KUKA KRL program: MyProgram_256().src

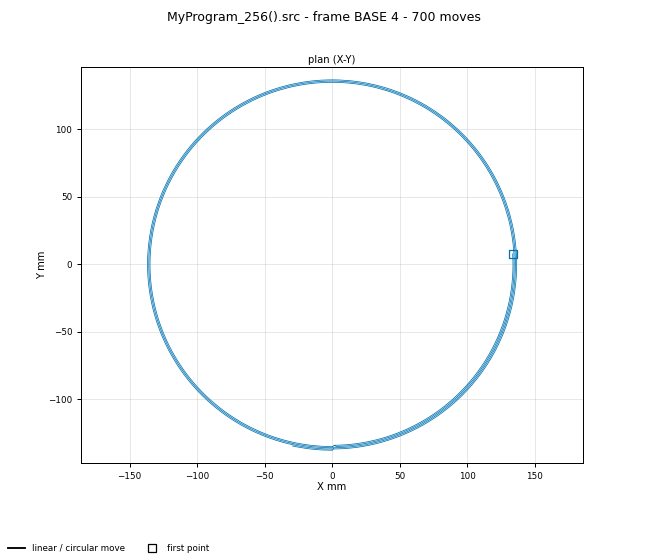
[picture p0: tool path of MyProgram_256().src in frame BASE 4, 700 of 700 moves have a stored position in this frame; points joined in program order, loops and branches not executed]
&ACCESS RVP
&REL 1
&PARAM TEMPLATE = C:\KRC\Roboter\Template\vorgabe
&PARAM EDITMASK = *
DEF MyProgram_256()
; ---- Setting reference (Base) ----
$BASE = BASE_DATA[4]

; --------------------------
; ---- Setting tool (TCP) ----
$TOOL = TOOL_DATA[3]
; --------------------------

$VEL.CP = VEL_APROX_PRINT
Startdeposition()
$VEL.CP = VEL_PRINT
LIN {X 133.7906,Y 7.8081,Z 166,A 3.583,B 11.1418,C 0.1363,E1 11.3023,E2 447.1439} C_DIS
LIN {X 133.9693,Y 3.6015,Z 166,A 1.8917,B 11.1418,C 0.1387,E1 11.3024,E2 448.8238} C_DIS
LIN {X 134.0189,Y -0.4124,Z 166,A 0.0697,B 11.1418,C 0.1466,E1 11.3024,E2 450.6604} C_DIS
LIN {X 133.9478,Y -4.3751,Z 166,A -1.598,B 11.1416,C 0.1508,E1 11.3024,E2 452.3268} C_DIS
LIN {X 133.7538,Y -8.4056,Z 166,A -3.1449,B 11.1416,C 0.1512,E1 11.3021,E2 453.8538} C_DIS
LIN {X 133.4765,Y -12.0532,Z 166,A -4.846,B 11.1416,C 0.1594,E1 11.3017,E2 455.5733} C_DIS
LIN {X 133.0684,Y -15.9212,Z 166,A -6.3681,B 11.1416,C 0.1606,E1 11.3012,E2 457.08} C_DIS
LIN {X 132.6216,Y -19.2954,Z 166,A -7.7805,B 11.1415,C 0.1637,E1 11.3007,E2 458.4888} C_DIS
LIN {X 131.994,Y -23.2035,Z 166,A -9.5019,B 11.1414,C 0.1694,E1 11.2999,E2 460.2156} C_DIS
LIN {X 131.3378,Y -26.6655,Z 166,A -10.9987,B 11.1414,C 0.1735,E1 11.2991,E2 461.7128} C_DIS
LIN {X 130.4251,Y -30.8268,Z 166,A -13.677,B 11.1409,C 0.2014,E1 11.2973,E2 464.497} C_DIS
LIN {X 128.7428,Y -37.2306,Z 166,A -15.3883,B 11.1412,C 0.18,E1 11.2961,E2 466.0757} C_DIS
LIN {X 127.5273,Y -41.2019,Z 166,A -17.6042,B 11.1409,C 0.1967,E1 11.2942,E2 468.3474} C_DIS
LIN {X 126.4482,Y -44.4042,Z 166,A -18.6879,B 11.141,C 0.1912,E1 11.2933,E2 469.3887} C_DIS
LIN {X 125.1769,Y -47.8735,Z 166,A -20.2354,B 11.141,C 0.1948,E1 11.2918,E2 470.9341} C_DIS
LIN {X 124.0766,Y -50.6551,Z 166,A -21.541,B 11.141,C 0.199,E1 11.2904,E2 472.2445} C_DIS
LIN {X 122.8258,Y -53.6156,Z 166,A -22.8653,B 11.1409,C 0.2015,E1 11.2889,E2 473.5642} C_DIS
LIN {X 120.5287,Y -58.6003,Z 166,A -25.1853,B 11.1408,C 0.2071,E1 11.2862,E2 475.8837} C_DIS
LIN {X 119.1646,Y -61.3246,Z 166,A -26.4556,B 11.1408,C 0.2098,E1 11.2846,E2 477.1515} C_DIS
LIN {X 117.7601,Y -63.9821,Z 166,A -27.884,B 11.1406,C 0.2169,E1 11.2827,E2 478.599} C_DIS
LIN {X 115.3948,Y -68.156,Z 166,A -29.8951,B 11.1405,C 0.2212,E1 11.2799,E2 480.6076} C_DIS
LIN {X 113.0597,Y -71.9634,Z 166,A -31.8065,B 11.1404,C 0.2262,E1 11.277,E2 482.5214} C_DIS
LIN {X 110.6658,Y -75.5929,Z 166,A -33.6473,B 11.1404,C 0.2303,E1 11.2742,E2 484.362} C_DIS
LIN {X 107.9816,Y -79.3793,Z 166,A -35.5798,B 11.1402,C 0.2339,E1 11.271,E2 486.2904} C_DIS
LIN {X 105.2313,Y -82.9912,Z 166,A -37.5088,B 11.1402,C 0.2382,E1 11.2677,E2 488.2202} C_DIS
LIN {X 101.0585,Y -88.0239,Z 166,A -40.4879,B 11.1399,C 0.2495,E1 11.2623,E2 491.2248} C_DIS
LIN {X 98.7885,Y -90.5647,Z 166,A -41.3605,B 11.1402,C 0.2376,E1 11.2608,E2 492.0274} C_DIS
LIN {X 93.0666,Y -96.4352,Z 166,A -44.9331,B 11.14,C 0.247,E1 11.2538,E2 495.6122} C_DIS
LIN {X 88.7789,Y -100.3962,Z 166,A -47.5027,B 11.1398,C 0.2542,E1 11.2485,E2 498.1936} C_DIS
LIN {X 83.3335,Y -104.9603,Z 166,A -50.5306,B 11.1397,C 0.2599,E1 11.242,E2 501.2236} C_DIS
LIN {X 79.6928,Y -107.7513,Z 166,A -52.6048,B 11.1395,C 0.2665,E1 11.2373,E2 503.3137} C_DIS
LIN {X 76.2597,Y -110.2074,Z 166,A -54.7708,B 11.1392,C 0.2789,E1 11.2323,E2 505.5257} C_DIS
LIN {X 72.8142,Y -112.5127,Z 166,A -56.0319,B 11.1394,C 0.269,E1 11.2295,E2 506.7259} C_DIS
LIN {X 70.1028,Y -114.2222,Z 166,A -57.527,B 11.1394,C 0.2744,E1 11.2259,E2 508.2376} C_DIS
LIN {X 66.5644,Y -116.3199,Z 166,A -59.1858,B 11.1394,C 0.2747,E1 11.2219,E2 509.8859} C_DIS
LIN {X 63.435,Y -118.0555,Z 166,A -60.712,B 11.1393,C 0.2769,E1 11.2181,E2 511.413} C_DIS
LIN {X 60.4507,Y -119.6095,Z 166,A -62.0754,B 11.1393,C 0.2771,E1 11.2148,E2 512.7684} C_DIS
LIN {X 57.3326,Y -121.1354,Z 166,A -63.5711,B 11.1392,C 0.2795,E1 11.211,E2 514.2669} C_DIS
LIN {X 54.3356,Y -122.5088,Z 166,A -64.9633,B 11.1392,C 0.2809,E1 11.2075,E2 515.6581} C_DIS
LIN {X 51.2255,Y -123.8416,Z 166,A -66.4225,B 11.1392,C 0.2831,E1 11.2037,E2 517.1201} C_DIS
LIN {X 48.4559,Y -124.9505,Z 166,A -67.7161,B 11.1391,C 0.285,E1 11.2003,E2 518.4169} C_DIS
LIN {X 44.8142,Y -126.3042,Z 166,A -69.8247,B 11.1387,C 0.298,E1 11.1947,E2 520.5818} C_DIS
LIN {X 40.9151,Y -127.6189,Z 166,A -71.2137,B 11.1389,C 0.2907,E1 11.1911,E2 521.9268} C_DIS
LIN {X 37.414,Y -128.6891,Z 166,A -73.2769,B 11.1386,C 0.3044,E1 11.1854,E2 524.052} C_DIS
LIN {X 32.597,Y -129.9931,Z 166,A -74.6609,B 11.139,C 0.2879,E1 11.1819,E2 525.3459} C_DIS
LIN {X 29.7032,Y -130.6843,Z 166,A -76.0129,B 11.139,C 0.2909,E1 11.1782,E2 526.7087} C_DIS
LIN {X 26.3148,Y -131.4091,Z 166,A -77.4611,B 11.1389,C 0.2911,E1 11.1742,E2 528.1538} C_DIS
LIN {X 23.6903,Y -131.9069,Z 166,A -78.6623,B 11.1389,C 0.2933,E1 11.1709,E2 529.363} C_DIS
LIN {X 20.3393,Y -132.4651,Z 166,A -80.0685,B 11.1389,C 0.2931,E1 11.167,E2 530.7645} C_DIS
LIN {X 16.9036,Y -132.9481,Z 166,A -81.7085,B 11.1387,C 0.2976,E1 11.1624,E2 532.4246} C_DIS
LIN {X 12.8845,Y -133.3967,Z 166,A -83.3725,B 11.1387,C 0.2968,E1 11.1578,E2 534.0817} C_DIS
LIN {X 9.0475,Y -133.7137,Z 166,A -85.082,B 11.1387,C 0.2989,E1 11.153,E2 535.8} C_DIS
LIN {X 4.8862,Y -133.9289,Z 166,A -86.7229,B 11.1387,C 0.296,E1 11.1485,E2 537.4245} C_DIS
LIN {X 0.9791,Y -134.0137,Z 166,A -87.7099,B 11.1392,C 0.28,E1 11.146,E2 538.3279} C_DIS
Enddeposition()
LIN {X 0.9791,Y -134.0137,Z 166,A -87.7099,B 11.1392,C 0.28,E1 11.146,E2 538.3279} C_DIS
Startdeposition()
$VEL.CP = VEL_PRINT
LIN {X 3.2943,Y -134.8946,Z 166,A -86.6554,B 11.0822,C 0.2874,E1 11.092,E2 537.3154} C_DIS
LIN {X 7.444,Y -134.7302,Z 166,A -84.8631,B 11.0822,C 0.2862,E1 11.097,E2 535.5186} C_DIS
LIN {X 11.3456,Y -134.4561,Z 166,A -83.3067,B 11.0822,C 0.2881,E1 11.1013,E2 533.9743} C_DIS
LIN {X 14.7948,Y -134.1208,Z 166,A -81.735,B 11.0822,C 0.285,E1 11.1057,E2 532.3891} C_DIS
LIN {X 18.5599,Y -133.6524,Z 166,A -80.1797,B 11.0822,C 0.2856,E1 11.11,E2 530.84} C_DIS
LIN {X 22.1578,Y -133.1021,Z 166,A -78.6595,B 11.0822,C 0.2853,E1 11.1142,E2 529.3219} C_DIS
LIN {X 26.1565,Y -132.3762,Z 166,A -76.8587,B 11.0823,C 0.2822,E1 11.1192,E2 527.5106} C_DIS
LIN {X 29.8744,Y -131.5852,Z 166,A -75.3332,B 11.0823,C 0.2832,E1 11.1233,E2 525.995} C_DIS
LIN {X 33.1445,Y -130.7996,Z 166,A -73.7747,B 11.0823,C 0.2787,E1 11.1276,E2 524.4191} C_DIS
LIN {X 38.4727,Y -129.334,Z 166,A -70.7758,B 11.0828,C 0.2601,E1 11.1359,E2 521.336} C_DIS
LIN {X 44.2696,Y -127.4648,Z 166,A -68.935,B 11.0825,C 0.2762,E1 11.1405,E2 519.5874} C_DIS
LIN {X 49.6533,Y -125.4682,Z 166,A -66.5654,B 11.0825,C 0.2751,E1 11.1466,E2 517.2246} C_DIS
LIN {X 53.2645,Y -123.976,Z 166,A -64.8895,B 11.0825,C 0.2726,E1 11.151,E2 515.5452} C_DIS
LIN {X 57.4577,Y -122.0912,Z 166,A -62.8633,B 11.0827,C 0.2681,E1 11.1561,E2 513.5079} C_DIS
LIN {X 61.1579,Y -120.2778,Z 166,A -61.2251,B 11.0827,C 0.2684,E1 11.1602,E2 511.8822} C_DIS
LIN {X 64.7709,Y -118.3737,Z 166,A -59.4725,B 11.0827,C 0.2653,E1 11.1645,E2 510.1257} C_DIS
LIN {X 68.6942,Y -116.1415,Z 166,A -57.6684,B 11.0827,C 0.2653,E1 11.1688,E2 508.334} C_DIS
LIN {X 72.9984,Y -113.4851,Z 166,A -55.0485,B 11.0831,C 0.2494,E1 11.1752,E2 505.6525} C_DIS
LIN {X 76.5356,Y -111.1302,Z 166,A -53.6572,B 11.0829,C 0.2569,E1 11.1783,E2 504.3116} C_DIS
LIN {X 78.8554,Y -109.4969,Z 166,A -52.2038,B 11.0831,C 0.2483,E1 11.1816,E2 502.8257} C_DIS
LIN {X 81.6626,Y -107.4193,Z 166,A -50.9427,B 11.0831,C 0.2513,E1 11.1844,E2 501.5911} C_DIS
LIN {X 85.2525,Y -104.5926,Z 166,A -49.0521,B 11.0831,C 0.2488,E1 11.1885,E2 499.7047} C_DIS
LIN {X 88.9879,Y -101.434,Z 166,A -46.5816,B 11.0834,C 0.2343,E1 11.1938,E2 497.1824} C_DIS
LIN {X 92.2495,Y -98.4766,Z 166,A -45.1583,B 11.0832,C 0.2422,E1 11.1966,E2 495.8134} C_DIS
LIN {X 97.1282,Y -93.6683,Z 166,A -42.264,B 11.0834,C 0.2363,E1 11.2023,E2 492.9179} C_DIS
LIN {X 104.1946,Y -85.7394,Z 166,A -37.7832,B 11.0836,C 0.2268,E1 11.2106,E2 488.4361} C_DIS
LIN {X 106.9401,Y -82.2894,Z 166,A -35.9194,B 11.0836,C 0.2225,E1 11.2138,E2 486.5713} C_DIS
LIN {X 109.6131,Y -78.6932,Z 166,A -34.07,B 11.0837,C 0.2193,E1 11.2168,E2 484.7265} C_DIS
LIN {X 112.0482,Y -75.1856,Z 166,A -32.2399,B 11.0838,C 0.2143,E1 11.2197,E2 482.8922} C_DIS
LIN {X 114.4423,Y -71.4883,Z 166,A -30.4055,B 11.0838,C 0.2105,E1 11.2224,E2 481.0602} C_DIS
LIN {X 116.8454,Y -67.4889,Z 166,A -28.4762,B 11.084,C 0.2068,E1 11.2251,E2 479.1352} C_DIS
LIN {X 119.0573,Y -63.5067,Z 166,A -26.6472,B 11.084,C 0.2045,E1 11.2276,E2 477.3172} C_DIS
LIN {X 120.8288,Y -60.0633,Z 166,A -25.0143,B 11.084,C 0.2004,E1 11.2296,E2 475.6837} C_DIS
LIN {X 122.3657,Y -56.8659,Z 166,A -23.4203,B 11.0842,C 0.1939,E1 11.2315,E2 474.077} C_DIS
LIN {X 124.3117,Y -52.4778,Z 166,A -21.4551,B 11.0842,C 0.1903,E1 11.2337,E2 472.1187} C_DIS
LIN {X 125.397,Y -49.8305,Z 166,A -19.8941,B 11.0845,C 0.1776,E1 11.2354,E2 470.5129} C_DIS
LIN {X 126.8018,Y -46.1359,Z 166,A -18.7424,B 11.0843,C 0.1871,E1 11.2364,E2 469.4254} C_DIS
LIN {X 128.0668,Y -42.497,Z 166,A -17.0395,B 11.0844,C 0.1807,E1 11.238,E2 467.7122} C_DIS
LIN {X 129.3159,Y -38.5344,Z 166,A -15.1809,B 11.0845,C 0.1732,E1 11.2395,E2 465.8399} C_DIS
LIN {X 131.0199,Y -32.2697,Z 166,A -12.4407,B 11.0846,C 0.1657,E1 11.2414,E2 463.0987} C_DIS
LIN {X 132.0233,Y -27.8806,Z 166,A -10.616,B 11.0846,C 0.1625,E1 11.2425,E2 461.2827} C_DIS
LIN {X 132.6854,Y -24.5424,Z 166,A -9.1493,B 11.0847,C 0.1578,E1 11.2433,E2 459.8117} C_DIS
LIN {X 133.3765,Y -20.4421,Z 166,A -7.5048,B 11.0847,C 0.1559,E1 11.244,E2 458.1803} C_DIS
LIN {X 133.9607,Y -16.1777,Z 166,A -5.7189,B 11.0848,C 0.1516,E1 11.2446,E2 456.3976} C_DIS
LIN {X 134.3488,Y -12.557,Z 166,A -4.1158,B 11.0849,C 0.1456,E1 11.2451,E2 454.7859} C_DIS
LIN {X 134.6817,Y -8.2474,Z 166,A -2.3861,B 11.0849,C 0.143,E1 11.2454,E2 453.0673} C_DIS
LIN {X 134.8728,Y -4.0791,Z 166,A -0.6094,B 11.085,C 0.1377,E1 11.2456,E2 451.2882} C_DIS
LIN {X 134.9378,Y -0.04,Z 166,A 1.162,B 11.085,C 0.1311,E1 11.2456,E2 449.5082} C_DIS
LIN {X 134.8901,Y 3.4547,Z 166,A 2.489,B 11.085,C 0.131,E1 11.2456,E2 448.199} C_DIS
LIN {X 134.7486,Y 7.0766,Z 166,A 4.1116,B 11.0852,C 0.1242,E1 11.2454,E2 446.5645} C_DIS
LIN {X 134.4614,Y 11.2831,Z 166,A 5.8418,B 11.0852,C 0.1206,E1 11.245,E2 444.8399} C_DIS
LIN {X 134.0572,Y 15.3692,Z 166,A 7.6181,B 11.0852,C 0.1146,E1 11.2445,E2 443.0579} C_DIS
LIN {X 133.5718,Y 19.1238,Z 166,A 9.1612,B 11.0853,C 0.1117,E1 11.2439,E2 441.5213} C_DIS
LIN {X 132.8726,Y 23.4966,Z 166,A 10.9743,B 11.0853,C 0.1081,E1 11.2431,E2 439.7147} C_DIS
LIN {X 132.2347,Y 26.8532,Z 166,A 12.3918,B 11.0853,C 0.1048,E1 11.2423,E2 438.3} C_DIS
LIN {X 131.3642,Y 30.8415,Z 166,A 14.2061,B 11.0854,C 0.0977,E1 11.2412,E2 436.4742} C_DIS
LIN {X 130.4871,Y 34.3569,Z 166,A 15.6135,B 11.0854,C 0.0969,E1 11.2402,E2 435.0815} C_DIS
LIN {X 127.8562,Y 43.1294,Z 166,A 19.4437,B 11.0855,C 0.0877,E1 11.2371,E2 431.2555} C_DIS
LIN {X 125.9505,Y 48.4128,Z 166,A 21.9343,B 11.0855,C 0.0783,E1 11.2346,E2 428.7501} C_DIS
LIN {X 124.6151,Y 51.7514,Z 166,A 23.2795,B 11.0855,C 0.079,E1 11.2332,E2 427.426} C_DIS
LIN {X 123.3051,Y 54.7996,Z 166,A 24.7105,B 11.0856,C 0.0747,E1 11.2316,E2 425.9913} C_DIS
LIN {X 121.9347,Y 57.7854,Z 166,A 25.9295,B 11.0856,C 0.0757,E1 11.2302,E2 424.7929} C_DIS
LIN {X 120.5504,Y 60.6224,Z 166,A 27.5633,B 11.0856,C 0.0644,E1 11.2281,E2 423.122} C_DIS
LIN {X 118.585,Y 64.3836,Z 166,A 29.2533,B 11.0856,C 0.0628,E1 11.2259,E2 421.4446} C_DIS
LIN {X 116.2237,Y 68.5543,Z 166,A 31.2775,B 11.0857,C 0.058,E1 11.2231,E2 419.4205} C_DIS
LIN {X 113.9119,Y 72.3311,Z 166,A 33.1854,B 11.0857,C 0.0526,E1 11.2203,E2 417.5079} C_DIS
LIN {X 111.4032,Y 76.1378,Z 166,A 35.1327,B 11.0857,C 0.0477,E1 11.2172,E2 415.5581} C_DIS
LIN {X 108.5416,Y 80.165,Z 166,A 37.1727,B 11.0857,C 0.0443,E1 11.2139,E2 413.524} C_DIS
LIN {X 105.4037,Y 84.2479,Z 166,A 39.3245,B 11.0857,C 0.0402,E1 11.2102,E2 411.3754} C_DIS
LIN {X 102.5505,Y 87.6991,Z 166,A 41.2143,B 11.0857,C 0.0363,E1 11.2068,E2 409.486} C_DIS
LIN {X 99.7635,Y 90.8563,Z 166,A 42.9515,B 11.0858,C 0.0338,E1 11.2036,E2 407.7542} C_DIS
LIN {X 96.7339,Y 94.0756,Z 166,A 44.8257,B 11.0858,C 0.03,E1 11.2,E2 405.8796} C_DIS
LIN {X 93.5509,Y 97.2419,Z 166,A 46.7346,B 11.0858,C 0.0261,E1 11.1961,E2 403.9697} C_DIS
LIN {X 90.4365,Y 100.1444,Z 166,A 48.4957,B 11.0858,C 0.0238,E1 11.1925,E2 402.2136} C_DIS
LIN {X 87.1345,Y 103.0304,Z 166,A 50.3568,B 11.0858,C 0.0203,E1 11.1886,E2 400.3521} C_DIS
LIN {X 82.6423,Y 106.6669,Z 166,A 52.7838,B 11.0858,C 0.0166,E1 11.1833,E2 397.9278} C_DIS
LIN {X 79.39,Y 109.1094,Z 166,A 54.717,B 11.0858,C 0.0085,E1 11.1789,E2 395.9689} C_DIS
LIN {X 76.6356,Y 111.0616,Z 166,A 55.9538,B 11.0858,C 0.0111,E1 11.1761,E2 394.7559} C_DIS
LIN {X 72.7812,Y 113.6243,Z 166,A 57.8669,B 11.0858,C 0.0094,E1 11.1716,E2 392.8489} C_DIS
LIN {X 70.1598,Y 115.262,Z 166,A 59.7231,B 11.0858,C -0.0062,E1 11.1671,E2 390.926} C_DIS
LIN {X 65.7435,Y 117.837,Z 166,A 61.3733,B 11.0858,C 0.0038,E1 11.1632,E2 389.3394} C_DIS
LIN {X 61.3017,Y 120.2046,Z 166,A 63.4284,B 11.0858,C 0.003,E1 11.1581,E2 387.294} C_DIS
LIN {X 57.4255,Y 122.1066,Z 166,A 65.3248,B 11.0858,C -0.0008,E1 11.1533,E2 385.39} C_DIS
LIN {X 53.8037,Y 123.7428,Z 166,A 66.8616,B 11.0858,C 0.001,E1 11.1495,E2 383.8714} C_DIS
LIN {X 51.0067,Y 124.9229,Z 166,A 68.2389,B 11.0858,C -0.0025,E1 11.1459,E2 382.4835} C_DIS
LIN {X 48.0838,Y 126.078,Z 166,A 69.5732,B 11.0858,C -0.0039,E1 11.1424,E2 381.1494} C_DIS
LIN {X 44.3701,Y 127.43,Z 166,A 71.2433,B 11.0858,C -0.0052,E1 11.138,E2 379.4803} C_DIS
LIN {X 40.5596,Y 128.6945,Z 166,A 72.9098,B 11.0858,C -0.0058,E1 11.1336,E2 377.8187} C_DIS
LIN {X 36.5064,Y 129.9015,Z 166,A 74.6137,B 11.0858,C -0.0049,E1 11.129,E2 376.1262} C_DIS
LIN {X 33.5563,Y 130.6951,Z 166,A 75.9903,B 11.0858,C -0.0077,E1 11.1253,E2 374.7403} C_DIS
LIN {X 29.219,Y 131.7344,Z 166,A 77.9192,B 11.0858,C -0.0097,E1 11.12,E2 372.8076} C_DIS
LIN {X 25.5308,Y 132.4966,Z 166,A 79.4037,B 11.0858,C -0.0078,E1 11.116,E2 371.3373} C_DIS
LIN {X 22.3336,Y 133.0728,Z 166,A 80.7898,B 11.0858,C -0.0086,E1 11.1122,E2 369.9507} C_DIS
LIN {X 19.4027,Y 133.5319,Z 166,A 82.129,B 11.0858,C -0.011,E1 11.1085,E2 368.6024} C_DIS
LIN {X 15.1101,Y 134.0869,Z 166,A 84.0114,B 11.0858,C -0.0126,E1 11.1032,E2 366.7153} C_DIS
LIN {X 11.1908,Y 134.4692,Z 166,A 85.5401,B 11.0858,C -0.0096,E1 11.099,E2 365.2045} C_DIS
LIN {X 7.4433,Y 134.7302,Z 166,A 87.1498,B 11.0858,C -0.0101,E1 11.0945,E2 363.5937} C_DIS
LIN {X 3.776,Y 134.8812,Z 166,A 88.7028,B 11.0858,C -0.0101,E1 11.0902,E2 362.0419} C_DIS
LIN {X 0.0512,Y 134.9359,Z 166,A 90.3904,B 11.0858,C -0.0125,E1 11.0855,E2 360.3424} C_DIS
LIN {X -4.3069,Y 134.8664,Z 166,A 92.2429,B 11.0858,C -0.0123,E1 11.0803,E2 358.4906} C_DIS
LIN {X -8.0812,Y 134.6919,Z 166,A 93.7983,B 11.0858,C -0.0109,E1 11.076,E2 356.9418} C_DIS
LIN {X -12.1781,Y 134.3852,Z 166,A 95.617,B 11.0858,C -0.012,E1 11.0709,E2 355.1151} C_DIS
LIN {X -15.9767,Y 133.9847,Z 166,A 97.1138,B 11.0858,C -0.0086,E1 11.0668,E2 353.6344} C_DIS
LIN {X -19.759,Y 133.481,Z 166,A 98.8468,B 11.0858,C -0.0104,E1 11.062,E2 351.8887} C_DIS
LIN {X -23.4175,Y 132.8867,Z 166,A 100.3617,B 11.0858,C -0.0082,E1 11.0578,E2 350.382} C_DIS
LIN {X -29.2343,Y 131.7311,Z 166,A 102.9727,B 11.0858,C -0.0087,E1 11.0507,E2 347.7615} C_DIS
LIN {X -32.8993,Y 130.8619,Z 166,A 104.4642,B 11.0858,C -0.005,E1 11.0466,E2 346.2841} C_DIS
LIN {X -40.2682,Y 128.7864,Z 166,A 107.7597,B 11.0858,C -0.0032,E1 11.0378,E2 342.9857} C_DIS
LIN {X -45.1128,Y 127.1707,Z 166,A 109.9932,B 11.0858,C -0.0025,E1 11.0319,E2 340.746} C_DIS
LIN {X -48.5595,Y 125.8935,Z 166,A 111.4862,B 11.0858,C 0.0007,E1 11.028,E2 339.2624} C_DIS
LIN {X -52.8416,Y 124.1588,Z 166,A 113.5616,B 11.0858,C 0.0005,E1 11.0226,E2 337.175} C_DIS
LIN {X -56.2955,Y 122.6295,Z 166,A 115.1651,B 11.0858,C 0.0025,E1 11.0185,E2 335.5728} C_DIS
LIN {X -59.9089,Y 120.905,Z 166,A 116.7903,B 11.0858,C 0.0064,E1 11.0145,E2 333.9581} C_DIS
LIN {X -62.7587,Y 119.4503,Z 166,A 118.4008,B 11.0858,C 0.0029,E1 11.0104,E2 332.3184} C_DIS
LIN {X -65.7148,Y 117.8529,Z 166,A 119.6761,B 11.0858,C 0.0083,E1 11.0074,E2 331.0628} C_DIS
LIN {X -69.5526,Y 115.6292,Z 166,A 121.5897,B 11.0858,C 0.0105,E1 11.0028,E2 329.1472} C_DIS
LIN {X -73.3631,Y 113.2495,Z 166,A 123.4696,B 11.0858,C 0.0142,E1 10.9983,E2 327.2726} C_DIS
LIN {X -76.9601,Y 110.8365,Z 166,A 125.3283,B 11.0858,C 0.0169,E1 10.9941,E2 325.4132} C_DIS
LIN {X -80.7021,Y 108.1424,Z 166,A 127.2863,B 11.0858,C 0.0204,E1 10.9897,E2 323.4571} C_DIS
LIN {X -84.0783,Y 105.5387,Z 166,A 129.0961,B 11.0858,C 0.0238,E1 10.9857,E2 321.6493} C_DIS
LIN {X -87.5106,Y 102.7107,Z 166,A 131.0342,B 11.0858,C 0.0264,E1 10.9815,E2 319.7071} C_DIS
LIN {X -90.8736,Y 99.7479,Z 166,A 132.9365,B 11.0858,C 0.0302,E1 10.9776,E2 317.8069} C_DIS
LIN {X -94.0356,Y 96.7726,Z 166,A 134.8016,B 11.0858,C 0.0336,E1 10.9738,E2 315.941} C_DIS
LIN {X -97.0207,Y 93.7793,Z 166,A 136.6156,B 11.0858,C 0.037,E1 10.9703,E2 314.1266} C_DIS
LIN {X -100.1248,Y 90.4582,Z 166,A 138.5869,B 11.0858,C 0.0404,E1 10.9665,E2 312.1524} C_DIS
LIN {X -102.9756,Y 87.199,Z 166,A 140.4235,B 11.0858,C 0.0446,E1 10.9632,E2 310.3181} C_DIS
LIN {X -105.8186,Y 83.7266,Z 166,A 142.3956,B 11.0858,C 0.0477,E1 10.9597,E2 308.3401} C_DIS
LIN {X -108.5448,Y 80.1605,Z 166,A 144.3194,B 11.0858,C 0.0518,E1 10.9565,E2 306.4162} C_DIS
LIN {X -111.1732,Y 76.4729,Z 166,A 146.2458,B 11.0858,C 0.0565,E1 10.9534,E2 304.4916} C_DIS
LIN {X -113.1011,Y 73.5916,Z 166,A 147.7031,B 11.0857,C 0.0604,E1 10.9512,E2 303.0376} C_DIS
LIN {X -116.3017,Y 68.4215,Z 166,A 150.8674,B 11.0857,C 0.0549,E1 10.9465,E2 299.8054} C_DIS
LIN {X -118.7385,Y 64.1002,Z 166,A 152.4844,B 11.0857,C 0.0706,E1 10.9445,E2 298.2505} C_DIS
LIN {X -120.7674,Y 60.1879,Z 166,A 154.1569,B 11.0856,C 0.0796,E1 10.9424,E2 296.6041} C_DIS
LIN {X -122.3681,Y 56.8608,Z 166,A 155.9282,B 11.0856,C 0.0796,E1 10.9402,E2 294.8099} C_DIS
LIN {X -124.2145,Y 52.7105,Z 166,A 157.9395,B 11.0856,C 0.0832,E1 10.938,E2 292.7909} C_DIS
LIN {X -125.6756,Y 49.12,Z 166,A 159.4782,B 11.0855,C 0.0899,E1 10.9364,E2 291.267} C_DIS
LIN {X -126.6749,Y 46.4878,Z 166,A 160.8447,B 11.0855,C 0.0898,E1 10.9351,E2 289.8812} C_DIS
LIN {X -127.8707,Y 43.0857,Z 166,A 162.2948,B 11.0855,C 0.0957,E1 10.9338,E2 288.4426} C_DIS
LIN {X -129.0062,Y 39.5536,Z 166,A 163.8233,B 11.0855,C 0.1011,E1 10.9325,E2 286.9215} C_DIS
LIN {X -130.1301,Y 35.6889,Z 166,A 165.5851,B 11.0854,C 0.1049,E1 10.9311,E2 285.1553} C_DIS
LIN {X -131.1109,Y 31.8923,Z 166,A 167.096,B 11.0853,C 0.1128,E1 10.9301,E2 283.6649} C_DIS
LIN {X -131.7353,Y 29.2141,Z 166,A 168.5191,B 11.0853,C 0.111,E1 10.9292,E2 282.2122} C_DIS
LIN {X -132.5032,Y 25.496,Z 166,A 170.0535,B 11.0853,C 0.1173,E1 10.9284,E2 280.6889} C_DIS
LIN {X -133.4542,Y 19.9402,Z 166,A 172.5073,B 11.0852,C 0.123,E1 10.9273,E2 278.2305} C_DIS
LIN {X -133.9559,Y 16.2178,Z 166,A 174.1522,B 11.0852,C 0.1266,E1 10.9267,E2 276.5812} C_DIS
LIN {X -134.3736,Y 12.2989,Z 166,A 175.9751,B 11.0852,C 0.1285,E1 10.9262,E2 274.7419} C_DIS
LIN {X -134.6956,Y 8.0211,Z 166,A 177.7364,B 11.085,C 0.1351,E1 10.9259,E2 272.9898} C_DIS
LIN {X -134.8823,Y 3.7362,Z 166,A 179.5485,B 11.085,C 0.1406,E1 10.9257,E2 271.1808} C_DIS
LIN {X -134.9356,Y -0.3613,Z 166,A -178.6024,B 11.085,C 0.1435,E1 10.9257,E2 269.3203} C_DIS
LIN {X -134.8611,Y -4.499,Z 166,A -176.8121,B 11.0849,C 0.148,E1 10.9258,E2 267.5277} C_DIS
LIN {X -134.6801,Y -8.2729,Z 166,A -175.32,B 11.0848,C 0.155,E1 10.926,E2 266.0509} C_DIS
LIN {X -134.3805,Y -12.227,Z 166,A -173.553,B 11.0848,C 0.1582,E1 10.9264,E2 264.2754} C_DIS
LIN {X -133.984,Y -15.9826,Z 166,A -171.9855,B 11.0847,C 0.1636,E1 10.9269,E2 262.7138} C_DIS
LIN {X -133.5215,Y -19.4759,Z 166,A -170.3404,B 11.0847,C 0.1649,E1 10.9276,E2 261.052} C_DIS
LIN {X -132.7568,Y -24.1437,Z 166,A -168.1585,B 11.0847,C 0.1671,E1 10.9286,E2 258.8507} C_DIS
LIN {X -131.6923,Y -29.4056,Z 166,A -166.0813,B 11.0844,C 0.1778,E1 10.9298,E2 256.8004} C_DIS
LIN {X -130.8854,Y -32.8066,Z 166,A -164.6481,B 11.0844,C 0.183,E1 10.9308,E2 255.3748} C_DIS
LIN {X -129.2705,Y -38.6896,Z 166,A -161.8793,B 11.0844,C 0.1866,E1 10.9329,E2 252.5865} C_DIS
LIN {X -128.0886,Y -42.4313,Z 166,A -160.3566,B 11.0842,C 0.1942,E1 10.9342,E2 251.0828} C_DIS
LIN {X -127.0144,Y -45.5462,Z 166,A -158.8651,B 11.0842,C 0.1961,E1 10.9356,E2 249.581} C_DIS
LIN {X -125.7973,Y -48.8068,Z 166,A -157.4493,B 11.0841,C 0.2014,E1 10.937,E2 248.174} C_DIS
LIN {X -124.6539,Y -51.6585,Z 166,A -156.0103,B 11.0841,C 0.2021,E1 10.9385,E2 246.7195} C_DIS
LIN {X -122.8621,Y -55.79,Z 166,A -153.5144,B 11.0841,C 0.1949,E1 10.9415,E2 244.153} C_DIS
LIN {X -120.7592,Y -60.2044,Z 166,A -151.916,B 11.0839,C 0.2103,E1 10.9434,E2 242.6153} C_DIS
LIN {X -118.9133,Y -63.7748,Z 166,A -150.2182,B 11.0839,C 0.2149,E1 10.9456,E2 240.9198} C_DIS
LIN {X -116.7533,Y -67.6479,Z 166,A -148.3442,B 11.0837,C 0.2198,E1 10.9481,E2 239.0482} C_DIS
LIN {X -114.5806,Y -71.2661,Z 166,A -146.76,B 11.0835,C 0.2285,E1 10.9504,E2 237.4907} C_DIS
LIN {X -110.5845,Y -77.3223,Z 166,A -143.3695,B 11.0835,C 0.2294,E1 10.9557,E2 234.0641} C_DIS
LIN {X -107.8991,Y -81.0275,Z 166,A -141.3804,B 11.0835,C 0.2328,E1 10.959,E2 232.0704} C_DIS
LIN {X -105.1542,Y -84.5589,Z 166,A -139.4806,B 11.0834,C 0.2371,E1 10.9623,E2 230.1715} C_DIS
LIN {X -102.335,Y -87.9496,Z 166,A -137.6022,B 11.0833,C 0.241,E1 10.9657,E2 228.2933} C_DIS
LIN {X -99.4392,Y -91.211,Z 166,A -135.7293,B 11.0832,C 0.2444,E1 10.9692,E2 226.4186} C_DIS
LIN {X -96.3548,Y -94.4634,Z 166,A -133.8083,B 11.0832,C 0.2479,E1 10.9729,E2 224.4963} C_DIS
LIN {X -93.2018,Y -97.5756,Z 166,A -131.9622,B 11.083,C 0.2524,E1 10.9766,E2 222.6552} C_DIS
LIN {X -90.1628,Y -100.3906,Z 166,A -130.1781,B 11.083,C 0.2551,E1 10.9803,E2 220.8686} C_DIS
LIN {X -83.2989,Y -106.155,Z 166,A -126.4596,B 11.0828,C 0.2639,E1 10.9883,E2 217.1623} C_DIS
LIN {X -80.1929,Y -108.521,Z 166,A -124.5877,B 11.0828,C 0.2619,E1 10.9925,E2 215.2643} C_DIS
LIN {X -76.3879,Y -111.2316,Z 166,A -122.6315,B 11.0828,C 0.2657,E1 10.997,E2 213.3119} C_DIS
LIN {X -72.2707,Y -113.95,Z 166,A -119.8748,B 11.083,C 0.2539,E1 11.0037,E2 210.4726} C_DIS
LIN {X -67.492,Y -116.8436,Z 166,A -118.3002,B 11.0825,C 0.2752,E1 11.0072,E2 208.9982} C_DIS
LIN {X -64.2292,Y -118.6689,Z 166,A -116.4925,B 11.0825,C 0.2723,E1 11.0117,E2 207.1633} C_DIS
LIN {X -60.62,Y -120.5516,Z 166,A -114.7418,B 11.0825,C 0.2739,E1 11.0161,E2 205.4098} C_DIS
LIN {X -56.7342,Y -122.4267,Z 166,A -113.091,B 11.0824,C 0.2801,E1 11.0202,E2 203.7816} C_DIS
LIN {X -54.0973,Y -123.6159,Z 166,A -111.7239,B 11.0824,C 0.2783,E1 11.0237,E2 202.3972} C_DIS
LIN {X -50.2533,Y -125.2266,Z 166,A -110.0539,B 11.0824,C 0.2823,E1 11.028,E2 200.7396} C_DIS
LIN {X -46.4533,Y -126.6874,Z 166,A -108.1905,B 11.0824,C 0.2808,E1 11.0329,E2 198.8592} C_DIS
LIN {X -42.5789,Y -128.0395,Z 166,A -106.6505,B 11.0822,C 0.2869,E1 11.0369,E2 197.3442} C_DIS
LIN {X -39.2946,Y -129.0855,Z 166,A -105.1159,B 11.0822,C 0.2864,E1 11.041,E2 195.8006} C_DIS
LIN {X -35.5277,Y -130.1747,Z 166,A -103.1997,B 11.0823,C 0.2816,E1 11.0463,E2 193.8528} C_DIS
LIN {X -30.8617,Y -131.3593,Z 166,A -101.2087,B 11.0823,C 0.284,E1 11.0517,E2 191.868} C_DIS
LIN {X -26.8049,Y -132.2446,Z 166,A -99.5925,B 11.0822,C 0.2883,E1 11.056,E2 190.2697} C_DIS
LIN {X -22.9646,Y -132.9675,Z 166,A -97.9179,B 11.0822,C 0.2886,E1 11.0606,E2 188.5927} C_DIS
LIN {X -19.3333,Y -133.5418,Z 166,A -96.3435,B 11.0822,C 0.2888,E1 11.065,E2 187.0162} C_DIS
LIN {X -15.689,Y -134.019,Z 166,A -94.7251,B 11.0822,C 0.2878,E1 11.0695,E2 185.39} C_DIS
LIN {X -11.3441,Y -134.4562,Z 166,A -92.9102,B 11.0822,C 0.289,E1 11.0745,E2 183.5793} C_DIS
LIN {X -7.2369,Y -134.7406,Z 166,A -91.0955,B 11.0822,C 0.2875,E1 11.0796,E2 181.7555} C_DIS
LIN {X -2.9261,Y -134.904,Z 166,A -89.2557,B 11.0822,C 0.2872,E1 11.0848,E2 179.914} C_DIS
LIN {X 0.9797,Y -134.9303,Z 166,A -88.3711,B 11.0817,C 0.3056,E1 11.087,E2 179.125} C_DIS
Enddeposition()
LIN {X 0.9797,Y -134.9303,Z 166,A -88.3711,B 11.0817,C 0.3056,E1 11.087,E2 179.125} C_DIS
Startdeposition()
$VEL.CP = VEL_PRINT
LIN {X 0,Y -135.8526,Z 166,A -88.6856,B 11.0291,C 0.3123,E1 11.0336,E2 179.4781} C_DIS
LIN {X -3.9166,Y -135.794,Z 166,A -90.4076,B 11.0291,C 0.3141,E1 11.0288,E2 181.2096} C_DIS
LIN {X -7.0843,Y -135.6658,Z 166,A -91.7269,B 11.0291,C 0.3136,E1 11.0251,E2 182.5272} C_DIS
LIN {X -10.6614,Y -135.4336,Z 166,A -93.1949,B 11.0291,C 0.3125,E1 11.021,E2 183.9904} C_DIS
LIN {X -13.7574,Y -135.1542,Z 166,A -94.5096,B 11.0291,C 0.3124,E1 11.0174,E2 185.3061} C_DIS
LIN {X -16.4181,Y -134.8549,Z 166,A -95.6334,B 11.0291,C 0.312,E1 11.0142,E2 186.4295} C_DIS
LIN {X -19.3516,Y -134.465,Z 166,A -96.9142,B 11.0291,C 0.3124,E1 11.0107,E2 187.7147} C_DIS
LIN {X -23.1444,Y -133.8666,Z 166,A -98.5188,B 11.0291,C 0.3115,E1 11.0063,E2 189.3182} C_DIS
LIN {X -25.7807,Y -133.3818,Z 166,A -99.6535,B 11.0291,C 0.3111,E1 11.0032,E2 190.4536} C_DIS
LIN {X -28.8496,Y -132.7516,Z 166,A -100.9929,B 11.0291,C 0.3109,E1 10.9995,E2 191.7955} C_DIS
LIN {X -32.627,Y -131.8764,Z 166,A -102.6213,B 11.0291,C 0.3099,E1 10.9951,E2 193.4236} C_DIS
LIN {X -35.2766,Y -131.1903,Z 166,A -103.7815,B 11.0292,C 0.3093,E1 10.9919,E2 194.5847} C_DIS
LIN {X -38.4456,Y -130.2968,Z 166,A -105.2074,B 11.0292,C 0.3092,E1 10.9881,E2 196.0154} C_DIS
LIN {X -42.1302,Y -129.1548,Z 166,A -106.811,B 11.0292,C 0.3074,E1 10.9838,E2 197.6164} C_DIS
LIN {X -44.771,Y -128.2609,Z 166,A -107.9934,B 11.0292,C 0.3066,E1 10.9807,E2 198.7996} C_DIS
LIN {X -47.9213,Y -127.1174,Z 166,A -109.421,B 11.0293,C 0.3056,E1 10.977,E2 200.2291} C_DIS
LIN {X -51.5725,Y -125.6829,Z 166,A -111.0781,B 11.0293,C 0.3041,E1 10.9727,E2 201.8867} C_DIS
LIN {X -54.6916,Y -124.3573,Z 166,A -112.5159,B 11.0293,C 0.3028,E1 10.969,E2 203.3257} C_DIS
LIN {X -57.54,Y -123.0637,Z 166,A -113.8445,B 11.0294,C 0.3015,E1 10.9656,E2 204.6553} C_DIS
LIN {X -60.8677,Y -121.4539,Z 166,A -115.4129,B 11.0294,C 0.2999,E1 10.9617,E2 206.2248} C_DIS
LIN {X -63.918,Y -119.8766,Z 166,A -116.7885,B 11.0296,C 0.2964,E1 10.9583,E2 207.5914} C_DIS
LIN {X -66.9388,Y -118.2164,Z 166,A -118.4582,B 11.0295,C 0.2993,E1 10.9541,E2 209.2877} C_DIS
LIN {X -70.6682,Y -116.0255,Z 166,A -120.2416,B 11.0295,C 0.2959,E1 10.9499,E2 211.0659} C_DIS
LIN {X -74.3398,Y -113.708,Z 166,A -122.1065,B 11.0296,C 0.2939,E1 10.9455,E2 212.9346} C_DIS
LIN {X -77.9473,Y -111.266,Z 166,A -123.9389,B 11.0296,C 0.2909,E1 10.9413,E2 214.7661} C_DIS
LIN {X -81.4845,Y -108.7023,Z 166,A -125.7938,B 11.0298,C 0.2882,E1 10.9371,E2 216.6221} C_DIS
LIN {X -84.9452,Y -106.02,Z 166,A -127.659,B 11.0298,C 0.2854,E1 10.933,E2 218.489} C_DIS
LIN {X -88.3235,Y -103.2224,Z 166,A -129.5252,B 11.0299,C 0.2824,E1 10.929,E2 220.3567} C_DIS
LIN {X -91.5587,Y -100.3637,Z 166,A -131.3706,B 11.0299,C 0.2795,E1 10.9252,E2 222.2045} C_DIS
LIN {X -94.8108,Y -97.2976,Z 166,A -133.3104,B 11.0301,C 0.277,E1 10.9213,E2 224.1504} C_DIS
LIN {X -97.9092,Y -94.1792,Z 166,A -135.1918,B 11.0301,C 0.2739,E1 10.9176,E2 226.0344} C_DIS
LIN {X -100.904,Y -90.9631,Z 166,A -137.0078,B 11.0302,C 0.2692,E1 10.9142,E2 227.8449} C_DIS
LIN {X -103.791,Y -87.6547,Z 166,A -138.9307,B 11.0303,C 0.2667,E1 10.9106,E2 229.7757} C_DIS
LIN {X -106.5658,Y -84.2594,Z 166,A -140.746,B 11.0304,C 0.2619,E1 10.9075,E2 231.5858} C_DIS
LIN {X -109.2247,Y -80.783,Z 166,A -142.6108,B 11.0305,C 0.2581,E1 10.9043,E2 233.452} C_DIS
LIN {X -111.7643,Y -77.2313,Z 166,A -144.5264,B 11.0305,C 0.2554,E1 10.9013,E2 235.3756} C_DIS
LIN {X -114.1815,Y -73.6104,Z 166,A -146.3683,B 11.0307,C 0.2511,E1 10.8984,E2 237.2171} C_DIS
LIN {X -116.4739,Y -69.9268,Z 166,A -148.1765,B 11.0307,C 0.2462,E1 10.8958,E2 239.0215} C_DIS
LIN {X -118.6392,Y -66.1866,Z 166,A -150.0191,B 11.0309,C 0.242,E1 10.8933,E2 240.8653} C_DIS
LIN {X -120.6757,Y -62.3963,Z 166,A -151.7848,B 11.0309,C 0.2364,E1 10.891,E2 242.6238} C_DIS
LIN {X -122.2112,Y -59.3325,Z 166,A -153.2466,B 11.0311,C 0.233,E1 10.8892,E2 244.0865} C_DIS
LIN {X -123.663,Y -56.244,Z 166,A -154.7022,B 11.0311,C 0.2296,E1 10.8875,E2 245.5431} C_DIS
LIN {X -124.8099,Y -53.645,Z 166,A -155.9194,B 11.0311,C 0.2268,E1 10.8861,E2 246.7616} C_DIS
LIN {X -126.3141,Y -50.0066,Z 166,A -157.5936,B 11.0313,C 0.2226,E1 10.8843,E2 248.4363} C_DIS
LIN {X -127.5134,Y -46.8642,Z 166,A -159.0288,B 11.0313,C 0.2191,E1 10.8829,E2 249.8724} C_DIS
LIN {X -128.4504,Y -44.2243,Z 166,A -160.2498,B 11.0313,C 0.2167,E1 10.8818,E2 251.0972} C_DIS
LIN {X -129.4944,Y -41.067,Z 166,A -161.6424,B 11.0315,C 0.2126,E1 10.8806,E2 252.4874} C_DIS
LIN {X -130.507,Y -37.7276,Z 166,A -163.1565,B 11.0315,C 0.2094,E1 10.8794,E2 254.0054} C_DIS
LIN {X -131.4743,Y -34.2115,Z 166,A -164.6884,B 11.0316,C 0.2049,E1 10.8783,E2 255.5353} C_DIS
LIN {X -132.4757,Y -30.0912,Z 166,A -166.5137,B 11.0316,C 0.2006,E1 10.8771,E2 257.3634} C_DIS
LIN {X -133.2829,Y -26.2982,Z 166,A -168.1528,B 11.0318,C 0.196,E1 10.8762,E2 259.0015} C_DIS
LIN {X -133.7741,Y -23.6611,Z 166,A -169.2973,B 11.0318,C 0.193,E1 10.8756,E2 260.1465} C_DIS
LIN {X -134.3607,Y -20.0752,Z 166,A -170.8496,B 11.0318,C 0.189,E1 10.8749,E2 261.6999} C_DIS
LIN {X -134.8711,Y -16.2824,Z 166,A -172.5012,B 11.032,C 0.1851,E1 10.8744,E2 263.3544} C_DIS
LIN {X -135.2329,Y -12.9371,Z 166,A -173.9484,B 11.032,C 0.1815,E1 10.8739,E2 264.8036} C_DIS
LIN {X -135.5092,Y -9.626,Z 166,A -175.3355,B 11.032,C 0.1771,E1 10.8736,E2 266.1876} C_DIS
LIN {X -135.6805,Y -6.7915,Z 166,A -176.5844,B 11.0321,C 0.1747,E1 10.8734,E2 267.4415} C_DIS
LIN {X -135.8053,Y -3.513,Z 166,A -177.9944,B 11.0321,C 0.1711,E1 10.8734,E2 268.8533} C_DIS
LIN {X -135.8545,Y 0,Z 166,A -179.5154,B 11.0322,C 0.1676,E1 10.8733,E2 270.3777} C_DIS
LIN {X -135.8053,Y 3.513,Z 166,A 178.9824,B 11.0322,C 0.1636,E1 10.8733,E2 271.8807} C_DIS
LIN {X -135.6658,Y 7.0843,Z 166,A 177.4669,B 11.0324,C 0.1594,E1 10.8736,E2 273.3956} C_DIS
LIN {X -135.4336,Y 10.6614,Z 166,A 175.9792,B 11.0324,C 0.1545,E1 10.8739,E2 274.8788} C_DIS
LIN {X -135.1542,Y 13.7574,Z 166,A 174.6472,B 11.0324,C 0.151,E1 10.8742,E2 276.212} C_DIS
LIN {X -134.8009,Y 16.8715,Z 166,A 173.3049,B 11.0325,C 0.1476,E1 10.8747,E2 277.5553} C_DIS
LIN {X -134.4455,Y 19.4876,Z 166,A 172.1734,B 11.0325,C 0.1447,E1 10.8751,E2 278.6878} C_DIS
LIN {X -133.8844,Y 23.0373,Z 166,A 170.636,B 11.0326,C 0.1407,E1 10.8758,E2 280.2263} C_DIS
LIN {X -133.3818,Y 25.7807,Z 166,A 169.4463,B 11.0326,C 0.1376,E1 10.8764,E2 281.4162} C_DIS
LIN {X -132.6454,Y 29.3416,Z 166,A 167.8992,B 11.0326,C 0.1334,E1 10.8773,E2 282.9633} C_DIS
LIN {X -131.8764,Y 32.627,Z 166,A 166.4391,B 11.0327,C 0.1301,E1 10.8783,E2 284.4263} C_DIS
LIN {X -131.1903,Y 35.2766,Z 166,A 165.2666,B 11.0327,C 0.1271,E1 10.8791,E2 285.5996} C_DIS
LIN {X -130.2968,Y 38.4456,Z 166,A 163.8449,B 11.0328,C 0.1239,E1 10.8802,E2 287.0237} C_DIS
LIN {X -129.1548,Y 42.1302,Z 166,A 162.207,B 11.0328,C 0.1195,E1 10.8816,E2 288.6612} C_DIS
LIN {X -128.0815,Y 45.2885,Z 166,A 160.7798,B 11.0328,C 0.116,E1 10.8829,E2 290.0893} C_DIS
LIN {X -126.9243,Y 48.4371,Z 166,A 159.3446,B 11.0329,C 0.1125,E1 10.8843,E2 291.5254} C_DIS
LIN {X -125.8156,Y 51.2433,Z 166,A 158.0303,B 11.0329,C 0.1098,E1 10.8857,E2 292.8433} C_DIS
LIN {X -124.3573,Y 54.6916,Z 166,A 156.453,B 11.0329,C 0.1055,E1 10.8874,E2 294.4186} C_DIS
LIN {X -123.1822,Y 57.2838,Z 166,A 155.2356,B 11.033,C 0.1026,E1 10.8888,E2 295.6366} C_DIS
LIN {X -121.7022,Y 60.3643,Z 166,A 153.7746,B 11.033,C 0.0991,E1 10.8906,E2 297.0984} C_DIS
LIN {X -120.1288,Y 63.4378,Z 166,A 152.3598,B 11.033,C 0.0944,E1 10.8924,E2 298.5065} C_DIS
LIN {X -118.2164,Y 66.9388,Z 166,A 150.4704,B 11.033,C 0.0944,E1 10.895,E2 300.4191} C_DIS
LIN {X -116.0255,Y 70.6682,Z 166,A 148.6773,B 11.0331,C 0.089,E1 10.8976,E2 302.2063} C_DIS
LIN {X -113.7949,Y 74.2059,Z 166,A 146.8706,B 11.0331,C 0.0855,E1 10.9003,E2 304.0162} C_DIS
LIN {X -111.266,Y 77.9473,Z 166,A 144.9632,B 11.0331,C 0.0808,E1 10.9033,E2 305.9218} C_DIS
LIN {X -108.7023,Y 81.4845,Z 166,A 143.0559,B 11.0332,C 0.0777,E1 10.9065,E2 307.8349} C_DIS
LIN {X -106.02,Y 84.9452,Z 166,A 141.231,B 11.0332,C 0.073,E1 10.9096,E2 309.6552} C_DIS
LIN {X -103.2224,Y 88.3235,Z 166,A 139.3604,B 11.0332,C 0.0692,E1 10.913,E2 311.5262} C_DIS
LIN {X -100.3216,Y 91.6051,Z 166,A 137.4922,B 11.0332,C 0.0655,E1 10.9165,E2 313.395} C_DIS
LIN {X -97.2976,Y 94.8108,Z 166,A 135.5601,B 11.0333,C 0.063,E1 10.9202,E2 315.3339} C_DIS
LIN {X -94.1792,Y 97.9092,Z 166,A 133.6879,B 11.0333,C 0.0595,E1 10.924,E2 317.2064} C_DIS
LIN {X -91.0751,Y 100.8024,Z 166,A 131.9187,B 11.0333,C 0.0554,E1 10.9276,E2 318.9713} C_DIS
LIN {X -87.6547,Y 103.791,Z 166,A 129.9486,B 11.0333,C 0.0528,E1 10.9318,E2 320.9459} C_DIS
LIN {X -84.2594,Y 106.5658,Z 166,A 128.1388,B 11.0333,C 0.0485,E1 10.9357,E2 322.7491} C_DIS
LIN {X -80.9114,Y 109.1291,Z 166,A 126.3268,B 11.0333,C 0.046,E1 10.9398,E2 324.5634} C_DIS
LIN {X -77.2313,Y 111.7643,Z 166,A 124.3678,B 11.0334,C 0.0438,E1 10.9442,E2 326.5266} C_DIS
LIN {X -73.6104,Y 114.1815,Z 166,A 122.5189,B 11.0334,C 0.041,E1 10.9486,E2 328.3753} C_DIS
LIN {X -69.9268,Y 116.4739,Z 166,A 120.7315,B 11.0334,C 0.0372,E1 10.9528,E2 330.1558} C_DIS
LIN {X -66.1866,Y 118.6392,Z 166,A 118.8976,B 11.0334,C 0.0347,E1 10.9573,E2 331.9895} C_DIS
LIN {X -62.3963,Y 120.6757,Z 166,A 117.1413,B 11.0334,C 0.0309,E1 10.9616,E2 333.7371} C_DIS
LIN {X -59.6895,Y 122.035,Z 166,A 115.8557,B 11.0334,C 0.0293,E1 10.9648,E2 335.0225} C_DIS
LIN {X -56.244,Y 123.663,Z 166,A 114.2415,B 11.0334,C 0.0274,E1 10.9689,E2 336.6363} C_DIS
LIN {X -53.645,Y 124.8099,Z 166,A 113.038,B 11.0334,C 0.0261,E1 10.972,E2 337.8394} C_DIS
LIN {X -50.5201,Y 126.1071,Z 166,A 111.5857,B 11.0334,C 0.025,E1 10.9757,E2 339.2935} C_DIS
LIN {X -46.8642,Y 127.5134,Z 166,A 109.946,B 11.0334,C 0.0229,E1 10.98,E2 340.9305} C_DIS
LIN {X -43.7114,Y 128.6283,Z 166,A 108.5308,B 11.0334,C 0.0216,E1 10.9837,E2 342.3452} C_DIS
LIN {X -41.067,Y 129.4944,Z 166,A 107.3541,B 11.0334,C 0.0205,E1 10.9868,E2 343.5213} C_DIS
LIN {X -37.3809,Y 130.6085,Z 166,A 105.725,B 11.0334,C 0.0192,E1 10.9912,E2 345.1499} C_DIS
LIN {X -33.1786,Y 131.7364,Z 166,A 103.8819,B 11.0334,C 0.0179,E1 10.9962,E2 346.9926} C_DIS
LIN {X -29.46,Y 132.6199,Z 166,A 102.2711,B 11.0334,C 0.0168,E1 11.0006,E2 348.6022} C_DIS
LIN {X -26.2982,Y 133.2829,Z 166,A 100.9064,B 11.0334,C 0.016,E1 11.0043,E2 349.9663} C_DIS
LIN {X -23.6611,Y 133.7741,Z 166,A 99.7743,B 11.0334,C 0.0153,E1 11.0074,E2 351.0977} C_DIS
LIN {X -20.0013,Y 134.3721,Z 166,A 98.2088,B 11.0334,C 0.0146,E1 11.0117,E2 352.6624} C_DIS
LIN {X -15.8236,Y 134.9259,Z 166,A 96.4582,B 11.0334,C 0.0132,E1 11.0166,E2 354.4087} C_DIS
LIN {X -12.9513,Y 135.2316,Z 166,A 95.2048,B 11.0334,C 0.0136,E1 11.0201,E2 355.6657} C_DIS
LIN {X -9.626,Y 135.5092,Z 166,A 93.8069,B 11.0334,C 0.013,E1 11.0239,E2 357.0617} C_DIS
LIN {X -6.0563,Y 135.7175,Z 166,A 92.2996,B 11.0334,C 0.0127,E1 11.0281,E2 358.5682} C_DIS
LIN {X -1.5044,Y 135.8442,Z 166,A 90.382,B 11.0334,C 0.0124,E1 11.0335,E2 360.4845} C_DIS
LIN {X 2.5199,Y 135.8273,Z 166,A 88.6356,B 11.0334,C 0.0135,E1 11.0384,E2 362.2359} C_DIS
LIN {X 6.0563,Y 135.7175,Z 166,A 87.1873,B 11.0334,C 0.0126,E1 11.0424,E2 363.6784} C_DIS
LIN {X 9.1209,Y 135.546,Z 166,A 85.8914,B 11.0334,C 0.0128,E1 11.046,E2 364.974} C_DIS
LIN {X 12.9116,Y 135.2354,Z 166,A 84.2598,B 11.0334,C 0.0137,E1 11.0506,E2 366.6082} C_DIS
LIN {X 16.3915,Y 134.8581,Z 166,A 82.7655,B 11.0334,C 0.0146,E1 11.0547,E2 368.1041} C_DIS
LIN {X 19.4876,Y 134.4455,Z 166,A 81.4907,B 11.0334,C 0.014,E1 11.0582,E2 369.3734} C_DIS
LIN {X 23.1444,Y 133.8666,Z 166,A 79.93,B 11.0334,C 0.0147,E1 11.0625,E2 370.9337} C_DIS
LIN {X 27.3217,Y 133.0746,Z 166,A 78.0822,B 11.0334,C 0.0169,E1 11.0676,E2 372.7874} C_DIS
LIN {X 30.5239,Y 132.3768,Z 166,A 76.7078,B 11.0334,C 0.0176,E1 11.0714,E2 374.1606} C_DIS
LIN {X 33.6919,Y 131.6062,Z 166,A 75.3844,B 11.0334,C 0.0172,E1 11.0749,E2 375.4775} C_DIS
LIN {X 36.8613,Y 130.7538,Z 166,A 74.0029,B 11.0334,C 0.0182,E1 11.0786,E2 376.8585} C_DIS
LIN {X 40.5483,Y 129.6602,Z 166,A 72.3854,B 11.0334,C 0.0194,E1 11.083,E2 378.4752} C_DIS
LIN {X 43.1922,Y 128.8012,Z 166,A 71.2153,B 11.0334,C 0.0203,E1 11.0861,E2 379.6448} C_DIS
LIN {X 46.4009,Y 127.6804,Z 166,A 69.7447,B 11.0334,C 0.0226,E1 11.0899,E2 381.1198} C_DIS
LIN {X 50.0066,Y 126.3141,Z 166,A 68.1664,B 11.0334,C 0.0231,E1 11.094,E2 382.6923} C_DIS
LIN {X 53.1343,Y 125.0307,Z 166,A 66.7461,B 11.0334,C 0.0245,E1 11.0977,E2 384.1119} C_DIS
LIN {X 55.7383,Y 123.8892,Z 166,A 65.5523,B 11.0334,C 0.0257,E1 11.1007,E2 385.305} C_DIS
LIN {X 58.827,Y 122.4527,Z 166,A 64.1217,B 11.0334,C 0.0273,E1 11.1044,E2 386.7348} C_DIS
LIN {X 61.8951,Y 120.9308,Z 166,A 62.6924,B 11.0334,C 0.0288,E1 11.1079,E2 388.1624} C_DIS
LIN {X 64.9241,Y 119.334,Z 166,A 61.1533,B 11.0334,C 0.0331,E1 11.1117,E2 389.7131} C_DIS
LIN {X 68.9384,Y 117.0609,Z 166,A 59.2761,B 11.0334,C 0.0341,E1 11.1163,E2 391.5823} C_DIS
LIN {X 72.385,Y 114.9616,Z 166,A 57.5267,B 11.0334,C 0.0379,E1 11.1204,E2 393.3377} C_DIS
LIN {X 76.2758,Y 112.4177,Z 166,A 55.637,B 11.0334,C 0.0392,E1 11.1248,E2 395.2191} C_DIS
LIN {X 79.603,Y 110.0869,Z 166,A 53.8777,B 11.0334,C 0.0432,E1 11.1288,E2 396.9844} C_DIS
LIN {X 83.3435,Y 107.2829,Z 166,A 51.9791,B 11.0334,C 0.0448,E1 11.133,E2 398.8746} C_DIS
LIN {X 86.5283,Y 104.7311,Z 166,A 50.2134,B 11.0334,C 0.049,E1 11.1368,E2 400.6462} C_DIS
LIN {X 89.8664,Y 101.8812,Z 166,A 48.3777,B 11.0334,C 0.0521,E1 11.1407,E2 402.4806} C_DIS
LIN {X 93.1139,Y 98.922,Z 166,A 46.5411,B 11.0334,C 0.0553,E1 11.1445,E2 404.3159} C_DIS
LIN {X 96.4221,Y 95.7001,Z 166,A 44.6559,B 11.0334,C 0.0576,E1 11.1482,E2 406.1943} C_DIS
LIN {X 99.5224,Y 92.4719,Z 166,A 42.8005,B 11.0334,C 0.0608,E1 11.1518,E2 408.0465} C_DIS
LIN {X 102.2613,Y 89.4337,Z 166,A 41.0345,B 11.0333,C 0.0655,E1 11.1551,E2 409.8183} C_DIS
LIN {X 105.2876,Y 85.8503,Z 166,A 39.1353,B 11.0333,C 0.0679,E1 11.1584,E2 411.7089} C_DIS
LIN {X 107.8178,Y 82.6502,Z 166,A 37.3927,B 11.0333,C 0.0724,E1 11.1614,E2 413.455} C_DIS
LIN {X 110.4216,Y 79.138,Z 166,A 35.5524,B 11.0333,C 0.0766,E1 11.1645,E2 415.296} C_DIS
LIN {X 113.0426,Y 75.3465,Z 166,A 33.6799,B 11.0333,C 0.0794,E1 11.1674,E2 417.1609} C_DIS
LIN {X 115.4217,Y 71.649,Z 166,A 31.8562,B 11.0332,C 0.0831,E1 11.1701,E2 418.982} C_DIS
LIN {X 117.4974,Y 68.1918,Z 166,A 30.1194,B 11.0332,C 0.0883,E1 11.1726,E2 420.7243} C_DIS
LIN {X 119.486,Y 64.6451,Z 166,A 28.3886,B 11.0331,C 0.0931,E1 11.1749,E2 422.4582} C_DIS
LIN {X 121.4539,Y 60.8677,Z 166,A 26.7467,B 11.0331,C 0.0937,E1 11.177,E2 424.0825} C_DIS
LIN {X 122.9465,Y 57.7934,Z 166,A 25.3242,B 11.0331,C 0.097,E1 11.1787,E2 425.5037} C_DIS
LIN {X 124.1789,Y 55.0906,Z 166,A 24.0548,B 11.0331,C 0.1007,E1 11.1801,E2 426.776} C_DIS
LIN {X 125.6829,Y 51.5725,Z 166,A 22.4956,B 11.0331,C 0.1036,E1 11.1818,E2 428.3298} C_DIS
LIN {X 126.9243,Y 48.4371,Z 166,A 21.0926,B 11.033,C 0.107,E1 11.1832,E2 429.7316} C_DIS
LIN {X 128.0815,Y 45.2885,Z 166,A 19.6976,B 11.033,C 0.1103,E1 11.1846,E2 431.1254} C_DIS
LIN {X 129.1548,Y 42.1302,Z 166,A 18.3099,B 11.033,C 0.1137,E1 11.1858,E2 432.5118} C_DIS
LIN {X 129.9858,Y 39.4842,Z 166,A 17.1077,B 11.0329,C 0.1178,E1 11.1868,E2 433.719} C_DIS
LIN {X 131.0517,Y 35.7963,Z 166,A 15.5609,B 11.0329,C 0.1205,E1 11.1879,E2 435.2583} C_DIS
LIN {X 132.1287,Y 31.5807,Z 166,A 13.7007,B 11.0328,C 0.1263,E1 11.1892,E2 437.1232} C_DIS
LIN {X 132.8494,Y 28.3969,Z 166,A 12.3573,B 11.0328,C 0.1293,E1 11.19,E2 438.4638} C_DIS
LIN {X 133.5238,Y 25.0377,Z 166,A 10.9898,B 11.0328,C 0.1314,E1 11.1907,E2 439.823} C_DIS
LIN {X 134.043,Y 22.0872,Z 166,A 9.6798,B 11.0327,C 0.1363,E1 11.1914,E2 441.1399} C_DIS
LIN {X 134.596,Y 18.4346,Z 166,A 8.1923,B 11.0327,C 0.139,E1 11.1919,E2 442.6204} C_DIS
LIN {X 135.1542,Y 13.7574,Z 166,A 6.2357,B 11.0326,C 0.1439,E1 11.1926,E2 444.5751} C_DIS
LIN {X 135.5092,Y 9.626,Z 166,A 4.5139,B 11.0326,C 0.1483,E1 11.1929,E2 446.2952} C_DIS
LIN {X 135.7175,Y 6.0563,Z 166,A 3.0283,B 11.0325,C 0.1522,E1 11.1932,E2 447.7796} C_DIS
LIN {X 135.8442,Y 1.5044,Z 166,A 1.2025,B 11.0325,C 0.1553,E1 11.1932,E2 449.5957} C_DIS
LIN {X 135.8273,Y -2.5199,Z 166,A -0.5849,B 11.0323,C 0.1627,E1 11.1932,E2 451.396} C_DIS
LIN {X 135.7175,Y -6.0563,Z 166,A -2.0142,B 11.0323,C 0.1654,E1 11.1931,E2 452.8191} C_DIS
LIN {X 135.546,Y -9.1209,Z 166,A -3.2935,B 11.0323,C 0.1688,E1 11.1929,E2 454.0979} C_DIS
LIN {X 135.1985,Y -13.2955,Z 166,A -5.0331,B 11.0321,C 0.1732,E1 11.1924,E2 455.8359} C_DIS
LIN {X 134.8671,Y -16.3163,Z 166,A -6.2964,B 11.0321,C 0.1765,E1 11.192,E2 457.0984} C_DIS
LIN {X 134.4455,Y -19.4876,Z 166,A -7.6406,B 11.0321,C 0.1803,E1 11.1915,E2 458.4434} C_DIS
LIN {X 133.8666,Y -23.1444,Z 166,A -9.1835,B 11.032,C 0.1844,E1 11.1908,E2 459.9857} C_DIS
LIN {X 133.3818,Y -25.7807,Z 166,A -10.3008,B 11.032,C 0.1873,E1 11.1903,E2 461.1026} C_DIS
LIN {X 132.6199,Y -29.46,Z 166,A -11.8662,B 11.0318,C 0.1914,E1 11.1893,E2 462.6675} C_DIS
LIN {X 131.8764,Y -32.627,Z 166,A -13.2222,B 11.0318,C 0.1949,E1 11.1885,E2 464.023} C_DIS
LIN {X 131.1903,Y -35.2766,Z 166,A -14.3638,B 11.0318,C 0.1979,E1 11.1876,E2 465.1643} C_DIS
LIN {X 130.2968,Y -38.4456,Z 166,A -15.7729,B 11.0317,C 0.2024,E1 11.1865,E2 466.5774} C_DIS
LIN {X 129.1548,Y -42.1302,Z 166,A -17.3436,B 11.0316,C 0.2055,E1 11.1852,E2 468.1431} C_DIS
LIN {X 128.2609,Y -44.771,Z 166,A -18.5062,B 11.0316,C 0.2084,E1 11.1842,E2 469.3053} C_DIS
LIN {X 127.0768,Y -48.0297,Z 166,A -19.9847,B 11.0315,C 0.213,E1 11.1827,E2 470.7875} C_DIS
LIN {X 125.7062,Y -51.5146,Z 166,A -21.5042,B 11.0315,C 0.2157,E1 11.1812,E2 472.3013} C_DIS
LIN {X 124.3573,Y -54.6916,Z 166,A -22.9511,B 11.0313,C 0.2195,E1 11.1796,E2 473.7489} C_DIS
LIN {X 123.1822,Y -57.2838,Z 166,A -24.1383,B 11.0313,C 0.2224,E1 11.1782,E2 474.9356} C_DIS
LIN {X 121.7022,Y -60.3643,Z 166,A -25.5633,B 11.0313,C 0.2258,E1 11.1764,E2 476.3602} C_DIS
LIN {X 120.1527,Y -63.3922,Z 166,A -26.9303,B 11.0312,C 0.2279,E1 11.1747,E2 477.7205} C_DIS
LIN {X 118.2164,Y -66.9388,Z 166,A -28.7738,B 11.031,C 0.236,E1 11.1722,E2 479.5833} C_DIS
LIN {X 116.1056,Y -70.5359,Z 166,A -30.4891,B 11.031,C 0.2394,E1 11.1697,E2 481.2952} C_DIS
LIN {X 113.708,Y -74.3398,Z 166,A -32.4028,B 11.0308,C 0.2447,E1 11.1668,E2 483.2133} C_DIS
LIN {X 111.266,Y -77.9473,Z 166,A -34.1668,B 11.0308,C 0.2473,E1 11.164,E2 484.9701} C_DIS
LIN {X 108.7023,Y -81.4845,Z 166,A -35.9986,B 11.0307,C 0.2515,E1 11.161,E2 486.8027} C_DIS
LIN {X 106.02,Y -84.9452,Z 166,A -37.8168,B 11.0306,C 0.2552,E1 11.1579,E2 488.6194} C_DIS
LIN {X 103.2224,Y -88.3235,Z 166,A -39.6476,B 11.0305,C 0.259,E1 11.1546,E2 490.4498} C_DIS
LIN {X 100.3136,Y -91.6139,Z 166,A -41.4809,B 11.0304,C 0.2627,E1 11.1511,E2 492.2828} C_DIS
LIN {X 97.2976,Y -94.8108,Z 166,A -43.3701,B 11.0303,C 0.2677,E1 11.1475,E2 494.1784} C_DIS
LIN {X 94.1792,Y -97.9092,Z 166,A -45.2058,B 11.0302,C 0.2712,E1 11.1438,E2 496.0138} C_DIS
LIN {X 90.9631,Y -100.904,Z 166,A -46.9872,B 11.0302,C 0.2732,E1 11.1402,E2 497.7881} C_DIS
LIN {X 87.6547,Y -103.791,Z 166,A -48.8756,B 11.03,C 0.2778,E1 11.1361,E2 499.683} C_DIS
LIN {X 84.2594,Y -106.5658,Z 166,A -50.6537,B 11.03,C 0.2796,E1 11.1323,E2 501.4541} C_DIS
LIN {X 80.783,Y -109.2247,Z 166,A -52.4829,B 11.03,C 0.2826,E1 11.1282,E2 503.2831} C_DIS
LIN {X 77.2313,Y -111.7643,Z 166,A -54.3618,B 11.0298,C 0.2869,E1 11.1239,E2 505.1685} C_DIS
LIN {X 73.6104,Y -114.1815,Z 166,A -56.182,B 11.0298,C 0.2896,E1 11.1197,E2 506.9884} C_DIS
LIN {X 69.9268,Y -116.4739,Z 166,A -57.9326,B 11.0298,C 0.2906,E1 11.1155,E2 508.7309} C_DIS
LIN {X 66.2771,Y -118.5883,Z 166,A -59.7191,B 11.0296,C 0.2936,E1 11.1112,E2 510.52} C_DIS
LIN {X 62.3963,Y -120.6757,Z 166,A -61.484,B 11.0296,C 0.2939,E1 11.1068,E2 512.2749} C_DIS
LIN {X 59.3325,Y -122.2112,Z 166,A -62.9187,B 11.0296,C 0.2957,E1 11.1032,E2 513.7096} C_DIS
LIN {X 56.6629,Y -123.4693,Z 166,A -64.1909,B 11.0296,C 0.2981,E1 11.1,E2 514.9862} C_DIS
LIN {X 53.1343,Y -125.0307,Z 166,A -65.7704,B 11.0295,C 0.299,E1 11.096,E2 516.5612} C_DIS
LIN {X 50.0066,Y -126.3141,Z 166,A -67.1866,B 11.0295,C 0.3005,E1 11.0923,E2 517.9773} C_DIS
LIN {X 46.9965,Y -127.4638,Z 166,A -68.5219,B 11.0295,C 0.3015,E1 11.0888,E2 519.3108} C_DIS
LIN {X 43.7104,Y -128.6286,Z 166,A -69.998,B 11.0294,C 0.3032,E1 11.0849,E2 520.7888} C_DIS
LIN {X 41.067,Y -129.4944,Z 166,A -71.1636,B 11.0294,C 0.3042,E1 11.0818,E2 521.9542} C_DIS
LIN {X 37.6486,Y -130.5301,Z 166,A -72.6766,B 11.0294,C 0.3058,E1 11.0778,E2 523.4693} C_DIS
LIN {X 34.2115,Y -131.4743,Z 166,A -74.1569,B 11.0293,C 0.3066,E1 11.0738,E2 524.9479} C_DIS
LIN {X 31.5624,Y -132.1331,Z 166,A -75.3511,B 11.0293,C 0.3086,E1 11.0705,E2 526.1481} C_DIS
LIN {X 28.3969,Y -132.8494,Z 166,A -76.7127,B 11.0293,C 0.3094,E1 11.0668,E2 527.5097} C_DIS
LIN {X 24.7201,Y -133.5845,Z 166,A -78.2376,B 11.0293,C 0.3092,E1 11.0626,E2 529.0288} C_DIS
LIN {X 20.0013,Y -134.3721,Z 166,A -80.2467,B 11.0292,C 0.3101,E1 11.0571,E2 531.038} C_DIS
LIN {X 15.8236,Y -134.9259,Z 166,A -82.0639,B 11.0292,C 0.312,E1 11.052,E2 532.8613} C_DIS
LIN {X 12.7154,Y -135.2542,Z 166,A -83.3769,B 11.0292,C 0.3124,E1 11.0484,E2 534.1744} C_DIS
LIN {X 8.0892,Y -135.6096,Z 166,A -85.3263,B 11.0292,C 0.3129,E1 11.043,E2 536.1239} C_DIS
LIN {X 3.513,Y -135.8053,Z 166,A -87.2519,B 11.0291,C 0.3132,E1 11.0376,E2 538.0496} C_DIS
LIN {X 0.9848,Y -135.8471,Z 166,A -88.0754,B 11.0293,C 0.3076,E1 11.0354,E2 538.8434} C_DIS
Enddeposition()
LIN {X 0.9848,Y -135.8471,Z 166,A -88.0754,B 11.0293,C 0.3076,E1 11.0354,E2 538.8434} C_DIS
Startdeposition()
$VEL.CP = VEL_PRINT
LIN {X 1.481,Y -136.7608,Z 166,A -86.9104,B 10.9754,C 0.2934,E1 10.9847,E2 537.6077} C_DIS
LIN {X 5.8512,Y -136.6426,Z 166,A -85.4935,B 10.9751,C 0.303,E1 10.9884,E2 536.243} C_DIS
LIN {X 8.7814,Y -136.4851,Z 166,A -83.9095,B 10.9754,C 0.2939,E1 10.993,E2 534.613} C_DIS
LIN {X 12.8737,Y -136.1596,Z 166,A -82.5188,B 10.9752,C 0.3014,E1 10.9967,E2 533.2635} C_DIS
LIN {X 17.3889,Y -135.6573,Z 166,A -80.8306,B 10.9751,C 0.3058,E1 11.0013,E2 531.6015} C_DIS
LIN {X 20.5239,Y -135.2185,Z 166,A -79.3987,B 10.9751,C 0.3024,E1 11.0053,E2 530.1553} C_DIS
LIN {X 24.4377,Y -134.5661,Z 166,A -77.49,B 10.9754,C 0.2952,E1 11.0107,E2 528.214} C_DIS
LIN {X 29.2115,Y -133.611,Z 166,A -75.6818,B 10.9752,C 0.2995,E1 11.0155,E2 526.434} C_DIS
LIN {X 33.4763,Y -132.6064,Z 166,A -74.1042,B 10.9752,C 0.3045,E1 11.0197,E2 524.888} C_DIS
LIN {X 36.6473,Y -131.7653,Z 166,A -72.513,B 10.9752,C 0.2978,E1 11.0241,E2 523.2682} C_DIS
LIN {X 40.0333,Y -130.7761,Z 166,A -71.1017,B 10.9752,C 0.298,E1 11.0278,E2 521.8642} C_DIS
LIN {X 43.1573,Y -129.7787,Z 166,A -69.6737,B 10.9754,C 0.2953,E1 11.0317,E2 520.4283} C_DIS
LIN {X 46.2468,Y -128.7101,Z 166,A -68.3955,B 10.9754,C 0.2961,E1 11.035,E2 519.1606} C_DIS
LIN {X 49.2647,Y -127.5857,Z 166,A -67.0145,B 10.9754,C 0.2937,E1 11.0386,E2 517.7744} C_DIS
LIN {X 51.9884,Y -126.5023,Z 166,A -65.6263,B 10.9755,C 0.2881,E1 11.0423,E2 516.3648} C_DIS
LIN {X 55.5978,Y -124.9559,Z 166,A -64.1361,B 10.9755,C 0.2899,E1 11.046,E2 514.8929} C_DIS
LIN {X 58.063,Y -123.8315,Z 166,A -62.7669,B 10.9757,C 0.2824,E1 11.0496,E2 513.493} C_DIS
LIN {X 63.1688,Y -121.3051,Z 166,A -60.5938,B 10.9757,C 0.2844,E1 11.0549,E2 511.345} C_DIS
LIN {X 67.1028,Y -119.1755,Z 166,A -58.7294,B 10.9757,C 0.2818,E1 11.0595,E2 509.4802} C_DIS
LIN {X 70.7738,Y -117.0326,Z 166,A -57.1466,B 10.9757,C 0.2841,E1 11.0632,E2 507.9209} C_DIS
LIN {X 75.6586,Y -113.9362,Z 166,A -54.4756,B 10.9759,C 0.2736,E1 11.0696,E2 505.2161} C_DIS
LIN {X 79.2214,Y -111.4885,Z 166,A -52.6755,B 10.9759,C 0.2706,E1 11.0737,E2 503.4155} C_DIS
LIN {X 82.6984,Y -108.9344,Z 166,A -50.9583,B 10.976,C 0.2696,E1 11.0775,E2 501.708} C_DIS
LIN {X 85.9825,Y -106.3607,Z 166,A -49.2735,B 10.976,C 0.2679,E1 11.0812,E2 500.0294} C_DIS
LIN {X 88.9874,Y -103.8601,Z 166,A -47.7073,B 10.976,C 0.2665,E1 11.0845,E2 498.4707} C_DIS
LIN {X 91.5847,Y -101.5774,Z 166,A -46.0965,B 10.9762,C 0.2593,E1 11.0879,E2 496.8378} C_DIS
LIN {X 94.8682,Y -98.5175,Z 166,A -44.2357,B 10.9763,C 0.2558,E1 11.0917,E2 494.9774} C_DIS
LIN {X 98.1241,Y -95.2747,Z 166,A -42.3812,B 10.9763,C 0.2535,E1 11.0953,E2 493.1298} C_DIS
LIN {X 100.9202,Y -92.3081,Z 166,A -40.2016,B 10.9767,C 0.2371,E1 11.0996,E2 490.888} C_DIS
LIN {X 104.0743,Y -88.7363,Z 166,A -38.0307,B 10.9769,C 0.2278,E1 11.1035,E2 488.6924} C_DIS
LIN {X 107.7822,Y -84.1943,Z 166,A -36.3528,B 10.9766,C 0.2429,E1 11.1063,E2 487.1117} C_DIS
LIN {X 110.3072,Y -80.8573,Z 166,A -34.5761,B 10.9767,C 0.238,E1 11.1092,E2 485.33} C_DIS
LIN {X 112.8073,Y -77.3309,Z 166,A -32.7748,B 10.9768,C 0.2337,E1 11.1121,E2 483.5279} C_DIS
LIN {X 115.28,Y -73.5943,Z 166,A -30.896,B 10.9769,C 0.229,E1 11.115,E2 481.6467} C_DIS
LIN {X 117.4053,Y -70.154,Z 166,A -29.1997,B 10.977,C 0.2245,E1 11.1174,E2 479.9483} C_DIS
LIN {X 119.7489,Y -66.0743,Z 166,A -27.2752,B 10.977,C 0.2206,E1 11.1201,E2 478.0274} C_DIS
LIN {X 121.2502,Y -63.2733,Z 166,A -25.4759,B 10.9774,C 0.2044,E1 11.1225,E2 476.1668} C_DIS
LIN {X 123.3908,Y -58.9892,Z 166,A -24.2789,B 10.9771,C 0.2209,E1 11.1238,E2 475.0707} C_DIS
LIN {X 124.9438,Y -55.6249,Z 166,A -22.4848,B 10.9773,C 0.2102,E1 11.1259,E2 473.2442} C_DIS
LIN {X 126.5774,Y -51.8048,Z 166,A -20.8593,B 10.9773,C 0.2085,E1 11.1277,E2 471.6314} C_DIS
LIN {X 128.1242,Y -47.8461,Z 166,A -19.0466,B 10.9774,C 0.2027,E1 11.1295,E2 469.8125} C_DIS
LIN {X 129.2643,Y -44.6744,Z 166,A -17.7335,B 10.9774,C 0.2014,E1 11.1307,E2 468.5104} C_DIS
LIN {X 130.2505,Y -41.7119,Z 166,A -16.3788,B 10.9775,C 0.1964,E1 11.1319,E2 467.1483} C_DIS
LIN {X 131.2265,Y -38.5316,Z 166,A -15.0454,B 10.9775,C 0.1941,E1 11.1329,E2 465.821} C_DIS
LIN {X 132.1313,Y -35.3045,Z 166,A -13.6272,B 10.9777,C 0.1897,E1 11.134,E2 464.3994} C_DIS
LIN {X 132.9233,Y -32.1947,Z 166,A -12.2562,B 10.9777,C 0.1851,E1 11.1349,E2 463.0236} C_DIS
LIN {X 133.6978,Y -28.8094,Z 166,A -10.8481,B 10.9777,C 0.1822,E1 11.1358,E2 461.6197} C_DIS
LIN {X 134.5947,Y -24.2775,Z 166,A -8.6521,B 10.978,C 0.1695,E1 11.1369,E2 459.3886} C_DIS
LIN {X 135.1348,Y -21.0647,Z 166,A -7.5724,B 10.978,C 0.1732,E1 11.1374,E2 458.3435} C_DIS
LIN {X 135.7163,Y -16.9343,Z 166,A -5.7735,B 10.978,C 0.1667,E1 11.138,E2 456.5363} C_DIS
LIN {X 136.0466,Y -14.03,Z 166,A -4.4979,B 10.978,C 0.1618,E1 11.1384,E2 455.2529} C_DIS
LIN {X 136.4479,Y -9.3523,Z 166,A -2.7692,B 10.978,C 0.1625,E1 11.1388,E2 453.5522} C_DIS
LIN {X 136.7386,Y -2.8348,Z 166,A -0.1289,B 10.9782,C 0.157,E1 11.1391,E2 450.9209} C_DIS
LIN {X 136.72,Y 3.5862,Z 166,A 2.5753,B 10.9782,C 0.1487,E1 11.1391,E2 448.2122} C_DIS
LIN {X 136.4695,Y 9.0351,Z 166,A 5.0093,B 10.9784,C 0.138,E1 11.1386,E2 445.7573} C_DIS
LIN {X 136.1491,Y 12.9834,Z 166,A 6.6788,B 10.9784,C 0.1328,E1 11.1382,E2 444.0848} C_DIS
LIN {X 135.597,Y 17.8488,Z 166,A 8.5582,B 10.9784,C 0.1315,E1 11.1376,E2 442.2251} C_DIS
LIN {X 135.0657,Y 21.5108,Z 166,A 10.1859,B 10.9786,C 0.125,E1 11.1369,E2 440.5862} C_DIS
LIN {X 134.3311,Y 25.6956,Z 166,A 11.884,B 10.9786,C 0.122,E1 11.136,E2 438.8967} C_DIS
LIN {X 133.5001,Y 29.7217,Z 166,A 13.6757,B 10.9786,C 0.1153,E1 11.135,E2 437.0948} C_DIS
LIN {X 132.6302,Y 33.3824,Z 166,A 15.0979,B 10.9786,C 0.1149,E1 11.134,E2 435.6905} C_DIS
LIN {X 131.831,Y 36.4121,Z 166,A 16.256,B 10.9786,C 0.1154,E1 11.1332,E2 434.5507} C_DIS
LIN {X 130.9815,Y 39.3622,Z 166,A 17.7856,B 10.9788,C 0.1053,E1 11.132,E2 432.9894} C_DIS
LIN {X 129.8176,Y 43.0403,Z 166,A 19.2385,B 10.9788,C 0.1052,E1 11.1307,E2 431.5556} C_DIS
LIN {X 128.7929,Y 46.0171,Z 166,A 20.7376,B 10.9788,C 0.0967,E1 11.1293,E2 430.0328} C_DIS
LIN {X 127.0981,Y 50.5129,Z 166,A 22.6238,B 10.9788,C 0.0946,E1 11.1274,E2 428.161} C_DIS
LIN {X 125.8625,Y 53.5195,Z 166,A 24.0724,B 10.9789,C 0.0887,E1 11.1259,E2 426.7005} C_DIS
LIN {X 124.2076,Y 57.2497,Z 166,A 25.611,B 10.9789,C 0.0887,E1 11.1241,E2 425.182} C_DIS
LIN {X 122.8507,Y 60.1076,Z 166,A 26.9781,B 10.9789,C 0.0841,E1 11.1224,E2 423.8088} C_DIS
LIN {X 121.1909,Y 63.3863,Z 166,A 28.3842,B 10.9789,C 0.0837,E1 11.1206,E2 422.4183} C_DIS
LIN {X 118.8661,Y 67.6494,Z 166,A 30.517,B 10.979,C 0.076,E1 11.1177,E2 420.2719} C_DIS
LIN {X 116.4516,Y 71.7261,Z 166,A 32.4774,B 10.979,C 0.0717,E1 11.1149,E2 418.3133} C_DIS
LIN {X 114.0215,Y 75.5302,Z 166,A 34.3052,B 10.979,C 0.0688,E1 11.1121,E2 416.4922} C_DIS
LIN {X 111.5611,Y 79.1189,Z 166,A 36.1684,B 10.979,C 0.0634,E1 11.1091,E2 414.6229} C_DIS
LIN {X 109.0312,Y 82.57,Z 166,A 37.9541,B 10.9791,C 0.0594,E1 11.1062,E2 412.8371} C_DIS
LIN {X 106.1888,Y 86.1956,Z 166,A 39.8242,B 10.9791,C 0.0566,E1 11.1029,E2 410.9735} C_DIS
LIN {X 103.3709,Y 89.5555,Z 166,A 41.5595,B 10.9791,C 0.0553,E1 11.0998,E2 409.2499} C_DIS
LIN {X 99.704,Y 93.6203,Z 166,A 43.9324,B 10.9791,C 0.0483,E1 11.0953,E2 406.8661} C_DIS
LIN {X 96.588,Y 96.8318,Z 166,A 45.7911,B 10.9791,C 0.0449,E1 11.0917,E2 405.0088} C_DIS
LIN {X 93.2194,Y 100.0784,Z 166,A 47.7191,B 10.9791,C 0.0418,E1 11.0878,E2 403.0839} C_DIS
LIN {X 89.7505,Y 103.201,Z 166,A 49.3869,B 10.9791,C 0.0455,E1 11.0843,E2 401.4512} C_DIS
LIN {X 87.5164,Y 105.1027,Z 166,A 50.8514,B 10.9792,C 0.0372,E1 11.0812,E2 399.9571} C_DIS
LIN {X 84.1876,Y 107.7875,Z 166,A 52.6833,B 10.9792,C 0.033,E1 11.0771,E2 398.1197} C_DIS
LIN {X 80.5415,Y 110.5385,Z 166,A 54.5834,B 10.9792,C 0.0301,E1 11.0729,E2 396.2209} C_DIS
LIN {X 76.9338,Y 113.079,Z 166,A 56.3684,B 10.9792,C 0.0287,E1 11.0688,E2 394.4434} C_DIS
LIN {X 73.4148,Y 115.3949,Z 166,A 58.1277,B 10.9792,C 0.0261,E1 11.0647,E2 392.6845} C_DIS
LIN {X 69.8336,Y 117.5962,Z 166,A 59.891,B 10.9792,C 0.0234,E1 11.0604,E2 390.9206} C_DIS
LIN {X 65.8662,Y 119.8641,Z 166,A 61.8002,B 10.9792,C 0.0209,E1 11.0558,E2 389.0119} C_DIS
LIN {X 62.3177,Y 121.744,Z 166,A 63.4071,B 10.9792,C 0.0206,E1 11.0518,E2 387.4142} C_DIS
LIN {X 58.9599,Y 123.4048,Z 166,A 64.9104,B 10.9792,C 0.0203,E1 11.0481,E2 385.9189} C_DIS
LIN {X 56.0079,Y 124.7725,Z 166,A 66.1872,B 10.9792,C 0.0208,E1 11.0449,E2 384.6527} C_DIS
LIN {X 50.0315,Y 127.2877,Z 166,A 69.0872,B 10.9792,C 0.0134,E1 11.0373,E2 381.7303} C_DIS
LIN {X 46.5069,Y 128.6164,Z 166,A 70.5979,B 10.9792,C 0.0135,E1 11.0334,E2 380.228} C_DIS
LIN {X 43.4112,Y 129.6941,Z 166,A 71.9405,B 10.9792,C 0.013,E1 11.0298,E2 378.8894} C_DIS
LIN {X 40.0378,Y 130.7748,Z 166,A 73.392,B 10.9792,C 0.0126,E1 11.026,E2 377.4421} C_DIS
LIN {X 36.0486,Y 131.9327,Z 166,A 75.3622,B 10.9792,C 0.0057,E1 11.0206,E2 375.4438} C_DIS
LIN {X 31.7529,Y 133.0298,Z 166,A 77.0407,B 10.9792,C 0.0088,E1 11.0161,E2 373.7878} C_DIS
LIN {X 27.5849,Y 133.9562,Z 166,A 78.8045,B 10.9792,C 0.0084,E1 11.0113,E2 372.0275} C_DIS
LIN {X 24.7418,Y 134.5116,Z 166,A 80.4676,B 10.9792,C -0.003,E1 11.0066,E2 370.3092} C_DIS
LIN {X 20.5404,Y 135.216,Z 166,A 81.8759,B 10.9792,C 0.0054,E1 11.0028,E2 368.948} C_DIS
LIN {X 16.1773,Y 135.8066,Z 166,A 83.6097,B 10.9792,C 0.0074,E1 10.9981,E2 367.2284} C_DIS
LIN {X 13.0688,Y 136.1409,Z 166,A 85.0905,B 10.9792,C 0.003,E1 10.9939,E2 365.727} C_DIS
LIN {X 5.4455,Y 136.6584,Z 166,A 88.1381,B 10.9792,C 0.0063,E1 10.9855,E2 362.6997} C_DIS
LIN {X 1.3425,Y 136.7615,Z 166,A 89.7311,B 10.9792,C 0.0092,E1 10.9811,E2 361.123} C_DIS
LIN {X -2.9658,Y 136.7359,Z 166,A 91.8532,B 10.9792,C 0.002,E1 10.975,E2 358.9628} C_DIS
LIN {X -7.6483,Y 136.5548,Z 166,A 93.6407,B 10.9792,C 0.0064,E1 10.9701,E2 357.1979} C_DIS
LIN {X -11.372,Y 136.2932,Z 166,A 95.1922,B 10.9792,C 0.0071,E1 10.9658,E2 355.6487} C_DIS
LIN {X -15.7348,Y 135.8594,Z 166,A 97.0043,B 10.9792,C 0.0084,E1 10.9608,E2 353.8408} C_DIS
LIN {X -18.9552,Y 135.4473,Z 166,A 98.4492,B 10.9792,C 0.007,E1 10.9567,E2 352.3862} C_DIS
LIN {X -22.6251,Y 134.8823,Z 166,A 99.9729,B 10.9792,C 0.0085,E1 10.9526,E2 350.8674} C_DIS
LIN {X -26.784,Y 134.1192,Z 166,A 101.7063,B 10.9792,C 0.0105,E1 10.9478,E2 349.1398} C_DIS
LIN {X -29.6476,Y 133.5168,Z 166,A 103.0828,B 10.9792,C 0.0079,E1 10.944,E2 347.7457} C_DIS
LIN {X -33.537,Y 132.5909,Z 166,A 104.6476,B 10.9792,C 0.0116,E1 10.9398,E2 346.1955} C_DIS
LIN {X -36.9803,Y 131.6721,Z 166,A 106.1677,B 10.9792,C 0.0122,E1 10.9357,E2 344.6732} C_DIS
LIN {X -41.2288,Y 130.4048,Z 166,A 107.8138,B 10.9792,C 0.0187,E1 10.9314,E2 343.0543} C_DIS
LIN {X -46.3553,Y 128.671,Z 166,A 110.2313,B 10.9792,C 0.0176,E1 10.925,E2 340.6203} C_DIS
LIN {X -49.9988,Y 127.3004,Z 166,A 112.1949,B 10.9792,C 0.012,E1 10.9197,E2 338.6172} C_DIS
LIN {X -53.0089,Y 126.0761,Z 166,A 113.3248,B 10.9792,C 0.0187,E1 10.9169,E2 337.5168} C_DIS
LIN {X -57.1634,Y 124.2475,Z 166,A 115.1924,B 10.9792,C 0.0219,E1 10.9122,E2 335.6549} C_DIS
LIN {X -59.9386,Y 122.934,Z 166,A 116.6347,B 10.9792,C 0.0201,E1 10.9085,E2 334.1946} C_DIS
LIN {X -63.3778,Y 121.1954,Z 166,A 118.0381,B 10.9792,C 0.027,E1 10.9051,E2 332.8185} C_DIS
LIN {X -66.7898,Y 119.3514,Z 166,A 119.7963,B 10.9792,C 0.0265,E1 10.9007,E2 331.0455} C_DIS
LIN {X -70.2663,Y 117.3383,Z 166,A 121.4121,B 10.9792,C 0.0305,E1 10.8969,E2 329.4395} C_DIS
LIN {X -73.1238,Y 115.5789,Z 166,A 123.2744,B 10.9792,C 0.0228,E1 10.8923,E2 327.5224} C_DIS
LIN {X -76.4661,Y 113.3955,Z 166,A 124.6174,B 10.9792,C 0.0328,E1 10.8893,E2 326.2216} C_DIS
LIN {X -80.0654,Y 110.8835,Z 166,A 126.4421,B 10.9792,C 0.0363,E1 10.8852,E2 324.4004} C_DIS
LIN {X -84.455,Y 107.5775,Z 166,A 128.8547,B 10.9792,C 0.0381,E1 10.8798,E2 321.9765} C_DIS
LIN {X -88.9689,Y 103.8761,Z 166,A 131.3068,B 10.9792,C 0.0427,E1 10.8746,E2 319.5261} C_DIS
LIN {X -91.259,Y 101.8693,Z 166,A 132.9566,B 10.9792,C 0.0373,E1 10.871,E2 317.8315} C_DIS
LIN {X -94.4341,Y 98.9331,Z 166,A 134.4372,B 10.9792,C 0.0481,E1 10.8681,E2 316.3937} C_DIS
LIN {X -97.7569,Y 95.6513,Z 166,A 136.359,B 10.9792,C 0.053,E1 10.8643,E2 314.4782} C_DIS
LIN {X -100.9157,Y 92.313,Z 166,A 138.4979,B 10.9792,C 0.0527,E1 10.8602,E2 312.315} C_DIS
LIN {X -104.522,Y 88.2092,Z 166,A 140.652,B 10.9792,C 0.0607,E1 10.8564,E2 310.18} C_DIS
LIN {X -107.3436,Y 84.7527,Z 166,A 142.5518,B 10.9791,C 0.0644,E1 10.853,E2 308.2785} C_DIS
LIN {X -109.9917,Y 81.2867,Z 166,A 144.4209,B 10.9791,C 0.0679,E1 10.8499,E2 306.4063} C_DIS
LIN {X -112.7708,Y 77.3841,Z 166,A 146.3882,B 10.9791,C 0.0736,E1 10.8468,E2 304.4461} C_DIS
LIN {X -115.3132,Y 73.5424,Z 166,A 148.3664,B 10.9791,C 0.0774,E1 10.8437,E2 302.4641} C_DIS
LIN {X -117.7187,Y 69.6279,Z 166,A 150.3291,B 10.979,C 0.0816,E1 10.8409,E2 300.4989} C_DIS
LIN {X -119.9731,Y 65.6663,Z 166,A 152.2327,B 10.979,C 0.0866,E1 10.8383,E2 298.5982} C_DIS
LIN {X -121.7502,Y 62.3057,Z 166,A 153.7057,B 10.9789,C 0.0933,E1 10.8365,E2 297.1416} C_DIS
LIN {X -123.3122,Y 59.1537,Z 166,A 155.1605,B 10.9789,C 0.0976,E1 10.8347,E2 295.6908} C_DIS
LIN {X -124.4973,Y 56.6231,Z 166,A 156.58,B 10.9789,C 0.0957,E1 10.833,E2 294.2421} C_DIS
LIN {X -125.9538,Y 53.3018,Z 166,A 157.9533,B 10.9788,C 0.1028,E1 10.8315,E2 292.8884} C_DIS
LIN {X -127.7825,Y 48.7582,Z 166,A 160.1665,B 10.9788,C 0.1051,E1 10.8292,E2 290.6578} C_DIS
LIN {X -130.6413,Y 40.4739,Z 166,A 163.7919,B 10.9787,C 0.1164,E1 10.826,E2 287.0422} C_DIS
LIN {X -131.8601,Y 36.3084,Z 166,A 165.6901,B 10.9787,C 0.1199,E1 10.8245,E2 285.1362} C_DIS
LIN {X -132.901,Y 32.2874,Z 166,A 167.3714,B 10.9786,C 0.1261,E1 10.8234,E2 283.4641} C_DIS
LIN {X -133.6884,Y 28.8533,Z 166,A 168.8499,B 10.9786,C 0.1303,E1 10.8225,E2 281.9869} C_DIS
LIN {X -134.3733,Y 25.4747,Z 166,A 170.3823,B 10.9785,C 0.1327,E1 10.8217,E2 280.4452} C_DIS
LIN {X -135.1309,Y 21.0897,Z 166,A 172.2651,B 10.9785,C 0.1377,E1 10.8208,E2 278.5621} C_DIS
LIN {X -135.7161,Y 16.9353,Z 166,A 174.0897,B 10.9784,C 0.1415,E1 10.8202,E2 276.7312} C_DIS
LIN {X -136.0389,Y 14.1013,Z 166,A 175.2088,B 10.9784,C 0.1466,E1 10.8198,E2 275.6228} C_DIS
LIN {X -136.3986,Y 10.0285,Z 166,A 177.0222,B 10.9783,C 0.1495,E1 10.8194,E2 273.7987} C_DIS
LIN {X -136.6551,Y 5.5316,Z 166,A 178.8789,B 10.9782,C 0.1557,E1 10.8192,E2 271.9477} C_DIS
LIN {X -136.7547,Y 1.8684,Z 166,A -179.7102,B 10.9781,C 0.1627,E1 10.8191,E2 270.5538} C_DIS
LIN {X -136.7602,Y -1.5246,Z 166,A -178.0281,B 10.9781,C 0.1616,E1 10.8191,E2 268.8409} C_DIS
LIN {X -136.662,Y -5.3537,Z 166,A -176.4939,B 10.9781,C 0.1677,E1 10.8192,E2 267.317} C_DIS
LIN {X -136.4371,Y -9.5009,Z 166,A -174.7193,B 10.9779,C 0.1721,E1 10.8196,E2 265.5399} C_DIS
LIN {X -136.1494,Y -12.9799,Z 166,A -173.2741,B 10.9779,C 0.1767,E1 10.8199,E2 264.0983} C_DIS
LIN {X -135.7828,Y -16.3769,Z 166,A -171.7536,B 10.9779,C 0.179,E1 10.8204,E2 262.5681} C_DIS
LIN {X -135.1915,Y -20.6985,Z 166,A -169.9431,B 10.9777,C 0.1847,E1 10.8211,E2 260.7614} C_DIS
LIN {X -134.6235,Y -24.1168,Z 166,A -168.5,B 10.9777,C 0.189,E1 10.8218,E2 259.3207} C_DIS
LIN {X -133.8493,Y -28.1079,Z 166,A -166.6315,B 10.9777,C 0.1905,E1 10.8229,E2 257.4332} C_DIS
LIN {X -132.8707,Y -32.4131,Z 166,A -164.3663,B 10.9777,C 0.187,E1 10.8244,E2 255.1176} C_DIS
LIN {X -131.7408,Y -36.7349,Z 166,A -162.7304,B 10.9775,C 0.1972,E1 10.8256,E2 253.5129} C_DIS
LIN {X -130.3383,Y -41.4369,Z 166,A -160.9132,B 10.9773,C 0.2079,E1 10.827,E2 251.7272} C_DIS
LIN {X -128.4259,Y -47.0352,Z 166,A -158.2887,B 10.9773,C 0.2116,E1 10.8295,E2 249.0866} C_DIS
LIN {X -126.8354,Y -51.1647,Z 166,A -156.5293,B 10.9771,C 0.2186,E1 10.8313,E2 247.3404} C_DIS
LIN {X -125.5385,Y -54.2688,Z 166,A -155.1338,B 10.9771,C 0.2226,E1 10.8328,E2 245.9477} C_DIS
LIN {X -124.06,Y -57.5689,Z 166,A -153.6307,B 10.977,C 0.2269,E1 10.8345,E2 244.4472} C_DIS
LIN {X -122.8312,Y -60.1471,Z 166,A -152.3062,B 10.977,C 0.2273,E1 10.8361,E2 243.1076} C_DIS
LIN {X -121.2482,Y -63.2771,Z 166,A -150.9042,B 10.9768,C 0.2325,E1 10.8379,E2 241.715} C_DIS
LIN {X -119.3416,Y -66.8072,Z 166,A -149.0446,B 10.9768,C 0.2329,E1 10.8405,E2 239.8343} C_DIS
LIN {X -116.927,Y -70.9484,Z 166,A -147.0442,B 10.9768,C 0.238,E1 10.8433,E2 237.8362} C_DIS
LIN {X -114.525,Y -74.7643,Z 166,A -145.1032,B 10.9767,C 0.2415,E1 10.8462,E2 235.8898} C_DIS
LIN {X -111.9795,Y -78.5258,Z 166,A -143.2503,B 10.9765,C 0.247,E1 10.8492,E2 234.0442} C_DIS
LIN {X -109.491,Y -81.9598,Z 166,A -141.4331,B 10.9765,C 0.2502,E1 10.8522,E2 232.2229} C_DIS
LIN {X -106.8856,Y -85.3291,Z 166,A -139.6137,B 10.9764,C 0.2535,E1 10.8553,E2 230.4} C_DIS
LIN {X -104.8432,Y -87.8264,Z 166,A -138.1162,B 10.9764,C 0.2533,E1 10.858,E2 228.8849} C_DIS
LIN {X -101.5505,Y -91.6145,Z 166,A -136.1467,B 10.9762,C 0.2606,E1 10.8617,E2 226.9331} C_DIS
LIN {X -98.5751,Y -94.8087,Z 166,A -134.244,B 10.9762,C 0.2628,E1 10.8653,E2 225.0218} C_DIS
LIN {X -95.3751,Y -98.0268,Z 166,A -132.3285,B 10.9761,C 0.2662,E1 10.8691,E2 223.1052} C_DIS
LIN {X -92.2008,Y -101.0185,Z 166,A -130.6101,B 10.9759,C 0.2721,E1 10.8726,E2 221.4013} C_DIS
LIN {X -89.23,Y -103.6512,Z 166,A -128.8725,B 10.9759,C 0.2735,E1 10.8763,E2 219.6548} C_DIS
LIN {X -85.931,Y -106.4022,Z 166,A -127.0127,B 10.9759,C 0.2754,E1 10.8803,E2 217.7879} C_DIS
LIN {X -82.2691,Y -109.2583,Z 166,A -125.1078,B 10.9758,C 0.2796,E1 10.8845,E2 215.8887} C_DIS
LIN {X -78.9806,Y -111.6586,Z 166,A -123.3208,B 10.9758,C 0.2805,E1 10.8886,E2 214.0918} C_DIS
LIN {X -75.1366,Y -114.2806,Z 166,A -121.4031,B 10.9756,C 0.2842,E1 10.893,E2 212.1783} C_DIS
LIN {X -71.4253,Y -116.6362,Z 166,A -119.5443,B 10.9756,C 0.2865,E1 10.8975,E2 210.3176} C_DIS
LIN {X -67.5169,Y -118.9416,Z 166,A -117.5943,B 10.9756,C 0.2879,E1 10.9022,E2 208.3616} C_DIS
LIN {X -64.0344,Y -120.8506,Z 166,A -115.9939,B 10.9755,C 0.2915,E1 10.9061,E2 206.7693} C_DIS
LIN {X -60.8435,Y -122.4876,Z 166,A -114.4819,B 10.9755,C 0.2931,E1 10.9099,E2 205.2562} C_DIS
LIN {X -57.3205,Y -124.1748,Z 166,A -112.1916,B 10.9757,C 0.2799,E1 10.9159,E2 202.8826} C_DIS
LIN {X -52.419,Y -126.3225,Z 166,A -110.498,B 10.9754,C 0.2949,E1 10.9201,E2 201.2589} C_DIS
LIN {X -48.868,Y -127.74,Z 166,A -108.9286,B 10.9754,C 0.2972,E1 10.9241,E2 199.6936} C_DIS
LIN {X -45.2793,Y -129.0546,Z 166,A -107.5289,B 10.9751,C 0.3032,E1 10.9278,E2 198.3193} C_DIS
LIN {X -41.924,Y -130.1827,Z 166,A -105.8831,B 10.9752,C 0.3006,E1 10.9322,E2 196.6526} C_DIS
LIN {X -37.429,Y -131.5466,Z 166,A -103.9397,B 10.9752,C 0.3026,E1 10.9374,E2 194.712} C_DIS
LIN {X -33.8659,Y -132.5075,Z 166,A -102.2908,B 10.9752,C 0.3011,E1 10.9419,E2 193.0497} C_DIS
LIN {X -29.5331,Y -133.5416,Z 166,A -100.5777,B 10.9751,C 0.3057,E1 10.9465,E2 191.3557} C_DIS
LIN {X -26.7712,Y -134.1218,Z 166,A -99.0141,B 10.9753,C 0.2972,E1 10.9509,E2 189.7432} C_DIS
LIN {X -23.3401,Y -134.7624,Z 166,A -97.7421,B 10.9752,C 0.3023,E1 10.9543,E2 188.4951} C_DIS
LIN {X -19.3745,Y -135.3874,Z 166,A -96.1795,B 10.9751,C 0.3057,E1 10.9586,E2 186.9471} C_DIS
LIN {X -12.6419,Y -136.1819,Z 166,A -92.922,B 10.9753,C 0.2962,E1 10.9678,E2 183.6354} C_DIS
LIN {X -8.7271,Y -136.4884,Z 166,A -91.4118,B 10.9753,C 0.2995,E1 10.9719,E2 182.1417} C_DIS
LIN {X -5.5305,Y -136.6551,Z 166,A -90.5941,B 10.9749,C 0.3122,E1 10.9741,E2 181.3901} C_DIS
LIN {X 0.9738,Y -136.7546,Z 166,A -88.9265,B 10.9742,C 0.3374,E1 10.9785,E2 179.854} C_DIS
Enddeposition()
LIN {X 0.9738,Y -136.7546,Z 166,A -88.9266,B 10.9742,C 0.3374,E1 10.9785,E2 179.8542} C_DIS
Startdeposition()
$VEL.CP = VEL_PRINT
LIN {X 0.2296,Y -137.6841,Z 166,A -89.0656,B 10.9179,C 0.3424,E1 10.9219,E2 180.0248} C_DIS
LIN {X -4.4434,Y -137.6129,Z 166,A -90.4088,B 10.9184,C 0.3282,E1 10.9183,E2 181.293} C_DIS
LIN {X -7.0241,Y -137.504,Z 166,A -91.5505,B 10.9184,C 0.3297,E1 10.9151,E2 182.4436} C_DIS
LIN {X -11.4323,Y -137.2078,Z 166,A -93.3113,B 10.9184,C 0.3277,E1 10.9102,E2 184.1953} C_DIS
LIN {X -16.7798,Y -136.6571,Z 166,A -95.5763,B 10.9184,C 0.328,E1 10.9039,E2 186.4647} C_DIS
LIN {X -19.6503,Y -136.2737,Z 166,A -97.7354,B 10.9177,C 0.35,E1 10.8976,E2 188.7441} C_DIS
LIN {X -26.186,Y -135.1703,Z 166,A -99.8756,B 10.9182,C 0.3345,E1 10.8919,E2 190.8077} C_DIS
LIN {X -29.3667,Y -134.515,Z 166,A -100.944,B 10.9184,C 0.3272,E1 10.8891,E2 191.8407} C_DIS
Enddeposition()
END
